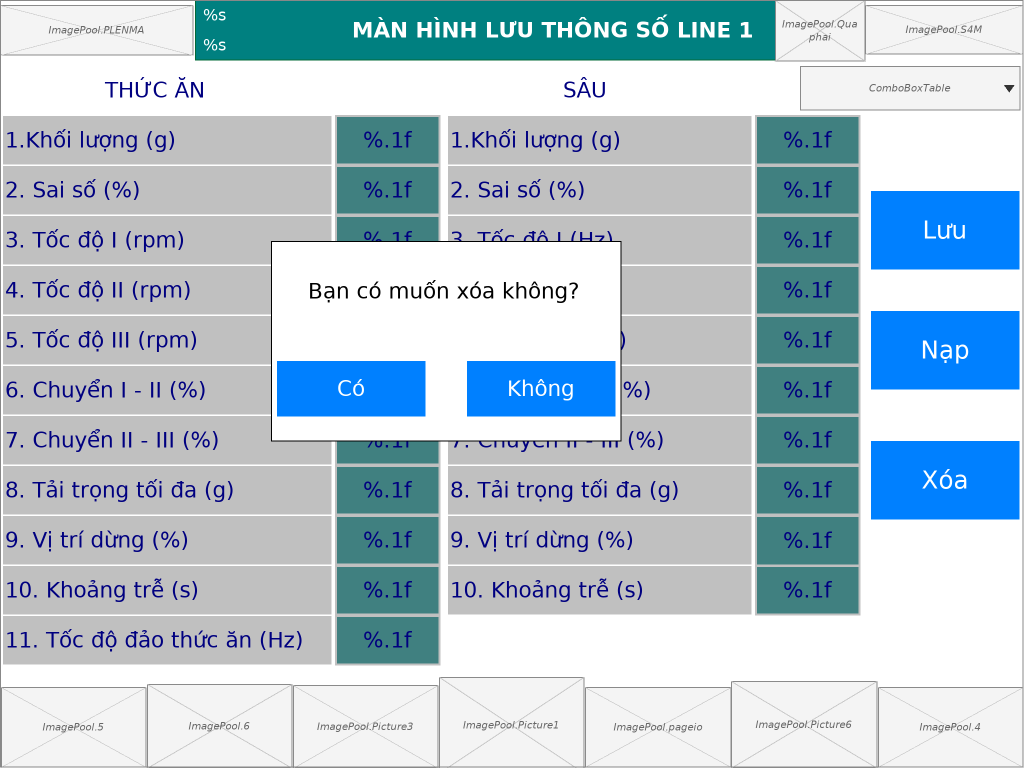
VISUALIZATION N_Recipe_Line1  // 1024x768
    Frame (0,687 1024x80)
        shows N_Footer_Line1()
    Frame (0,0 1024x60)
        shows N_Header()
    Textfield (353,5 400x50), "MÀN HÌNH LƯU THÔNG SỐ LINE 1"
    Textfield (80,75 150x30), "THỨC ĂN"
    Textfield (545,75 80x30), "SÂU"
    Rectangle (870,190 150x80), "Lưu"
        tap GVL_OF_VU.bRecSave[1]
        OnDialogClosed: execute { bSave1 := true; }
        OnMouseClick: write PRG_MainRecipe1.NameSave via VisuDialogs.Keypad
    Rectangle (870,440 150x80), "Xóa"
        tap GVL_OF_VU.bRecDelete[1]
        OnMouseDown: execute { GVL_OF_VU.bDeleteRecipe1 := TRUE; }
    Rectangle (870,310 150x80), "Nạp"
        tap GVL_OF_VU.bRecLoad[1]
        OnMouseDown: execute { bLoad1 := true; }
    ComboBoxTable (800,66 220x44), variable: PRG_MainRecipe1.RecipeNameIdx, data array: PRG_MainRecipe1.RecipeList
        p3854506369: PRG_MainRecipe1.RecipeList[INDEX]
    Rectangle (447,115 305x50), "1.Khối lượng (g)"
    Rectangle (447,165 305x50), "2. Sai số (%)"
    Rectangle (447,215 305x50), "3. Tốc độ I (Hz)"
    Rectangle (447,265 305x50), "4. Tốc độ II (Hz)"
    Rectangle (447,365 305x50), "6. Chuyển I - II (%)"
    Rectangle (447,465 305x50), "8. Tải trọng tối đa (g)"
    Rectangle (447,315 305x50), "5. Tốc độ III (Hz)"
    Rectangle (447,415 305x50), "7. Chuyển II - III (%)"
    Rectangle (447,565 305x50), "10. Khoảng trễ (s)"
    Rectangle (447,515 305x50), "9. Vị trí dừng (%)"
    Rectangle (2,115 330x50), "1.Khối lượng (g)"
    Rectangle (2,165 330x50), "2. Sai số (%)"
    Rectangle (2,215 330x50), "3. Tốc độ I (rpm)"
    Rectangle (2,265 330x50), "4. Tốc độ II (rpm)"
    Rectangle (2,365 330x50), "6. Chuyển I - II (%)"
    Rectangle (2,465 330x50), "8. Tải trọng tối đa (g)"
    Rectangle (2,315 330x50), "5. Tốc độ III (rpm)"
    Rectangle (2,415 330x50), "7. Chuyển II - III (%)"
    Rectangle (2,565 330x50), "10. Khoảng trễ (s)"
    Rectangle (2,515 330x50), "9. Vị trí dừng (%)"
    Rectangle (2,615 330x50), "11. Tốc độ đảo thức ăn (Hz)"
    Image (775,0 90x61), image: ImagePool.Qua phai
        OnMouseClick: change screen: N_Recipe_Line2
    Textfield (335,115 105x50), "%.1f", text variable: PR_Line01.fDerisedWeight_Food
    Textfield (335,165 105x50), "%.1f", text variable: PR_Line01.fDelta_Food
    Textfield (335,215 105x50), "%.1f", text variable: PR_Line01.fFast_Speed
    Textfield (335,265 105x50), "%.1f", text variable: PR_Line01.fSlow_Speed_1
    Textfield (335,315 105x50), "%.1f", text variable: PR_Line01.fSlow_Speed_2
    Textfield (335,365 105x50), "%.1f", text variable: PR_Line01.fChangeMode_Food_1
    Textfield (335,415 105x50), "%.1f", text variable: PR_Line01.fChangeMode_Food_2
    Textfield (335,465 105x50), "%.1f", text variable: PR_Line01.fMaxWeight_Food
    Textfield (335,515 105x50), "%.1f", text variable: PR_Line01.fPerStop_Food
    Textfield (335,565 105x50), "%.1f", text variable: PR_Line01.fTimer_Check_Food
    Textfield (335,615 105x50), "%.1f", text variable: PR_Line01.fSpeed_motor_mixer
    Textfield (755,115 105x50), "%.1f", text variable: PR_Line01.fDerisedWeight_Worm
    Textfield (755,165 105x50), "%.1f", text variable: PR_Line01.fDelta_Worm
    Textfield (755,215 105x50), "%.1f", text variable: PR_Line01.fFast_Speed_vibrating_funnel
    Textfield (755,265 105x50), "%.1f", text variable: PR_Line01.fSlow_Speed_vibrating_funnel_1
    Textfield (755,315 105x50), "%.1f", text variable: PR_Line01.fSlow_Speed_vibrating_funnel_2
    Textfield (755,365 105x50), "%.1f", text variable: PR_Line01.fChangeMode_Worm_1
    Textfield (755,415 105x50), "%.1f", text variable: PR_Line01.fChangeMode_Worm_2
    Textfield (755,465 105x50), "%.1f", text variable: PR_Line01.fMaxWeight_Worm
    Textfield (755,515 105x51), "%.1f", text variable: PR_Line01.fPerStop_Worm
    Textfield (755,565 105x50), "%.1f", text variable: PR_Line01.fTimer_Check_Worm
    GroupBox (271,241 350x200), invisible if: not GVL_OF_VU.bDeleteRecipe1, input disabled if: not GVL_OF_VU.bDeleteRecipe1
        Rectangle (0,0 350x200)
        Rectangle (5,119 150x57), "Có"
            OnMouseDown: execute { bDelete1 := true; }
            OnMouseUp: execute { GVL_OF_VU.bDeleteRecipe1 := FALSE; }
        Label (4,29 338x42), "Bạn có muốn xóa không?"
        Rectangle (195,119 150x57), "Không"
            OnMouseDown: execute { GVL_OF_VU.bDeleteRecipe1 := FALSE; }
END_VISUALIZATION

// ---- VISUs/Recipe/N_Recipe_Line2.TcVIS
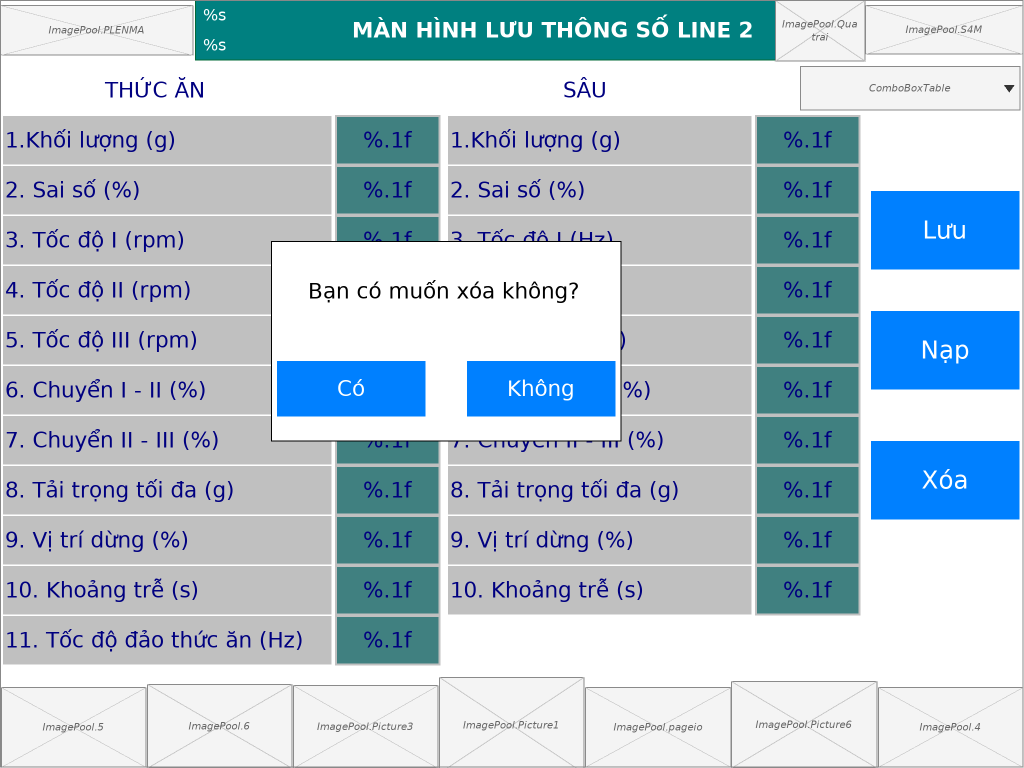
VISUALIZATION N_Recipe_Line2  // 1024x768
    Frame (0,687 1024x80)
        shows N_Footer_Line2()
    Frame (0,0 1024x60)
        shows N_Header()
    Textfield (353,5 400x50), "MÀN HÌNH LƯU THÔNG SỐ LINE 2"
    Textfield (80,75 150x30), "THỨC ĂN"
    Textfield (545,75 80x30), "SÂU"
    Rectangle (870,190 150x80), "Lưu"
        tap GVL_OF_VU.bRecSave[2]
        OnDialogClosed: execute { bSave2 := true; }
        OnMouseDown: write PRG_MainRecipe1_1.NameSave via VisuDialogs.Keypad
    Rectangle (870,440 150x80), "Xóa"
        tap GVL_OF_VU.bRecDelete[2]
        OnMouseClick: execute { GVL_OF_VU.bDeleteRecipe2 := true; }
    Rectangle (870,310 150x80), "Nạp"
        tap GVL_OF_VU.bRecLoad[2]
        OnMouseClick: execute { bLoad2 := true; }
    Group (447,115 305x500)
        Rectangle (0,0 305x50), "1.Khối lượng (g)"
        Rectangle (0,50 305x50), "2. Sai số (%)"
        Rectangle (0,100 305x50), "3. Tốc độ I (Hz)"
        Rectangle (0,150 305x50), "4. Tốc độ II (Hz)"
        Rectangle (0,250 305x50), "6. Chuyển I - II (%)"
        Rectangle (0,350 305x50), "8. Tải trọng tối đa (g)"
        Rectangle (0,200 305x50), "5. Tốc độ III (Hz)"
        Rectangle (0,300 305x50), "7. Chuyển II - III (%)"
        Rectangle (0,450 305x50), "10. Khoảng trễ (s)"
        Rectangle (0,400 305x50), "9. Vị trí dừng (%)"
    Textfield (755,115 105x50), "%.1f", text variable: PR_Line02.fDerisedWeight_Worm
    Textfield (755,165 105x50), "%.1f", text variable: PR_Line02.fDelta_Worm
    Textfield (755,215 105x50), "%.1f", text variable: PR_Line02.fFast_Speed_vibrating_funnel
    Textfield (755,265 105x50), "%.1f", text variable: PR_Line02.fSlow_Speed_vibrating_funnel_1
    Textfield (755,315 105x50), "%.1f", text variable: PR_Line02.fSlow_Speed_vibrating_funnel_2
    Textfield (755,365 105x50), "%.1f", text variable: PR_Line02.fChangeMode_Worm_1
    Textfield (755,415 105x50), "%.1f", text variable: PR_Line02.fChangeMode_Worm_2
        OnMouseDown: write GVL_OF_VU.fRecChangeII_IIIOfWorm[2] via VisuDialogs.Numpad
    Textfield (755,465 105x50), "%.1f", text variable: PR_Line02.fMaxWeight_Worm
    Textfield (755,515 105x50), "%.1f", text variable: PR_Line02.fPerStop_Worm
    Textfield (755,565 105x50), "%.1f", text variable: PR_Line02.fTimer_check_Worm
    Rectangle (2,115 330x50), "1.Khối lượng (g)"
    Rectangle (2,165 330x50), "2. Sai số (%)"
    Rectangle (2,215 330x50), "3. Tốc độ I (rpm)"
    Rectangle (2,265 330x50), "4. Tốc độ II (rpm)"
    Rectangle (2,365 330x50), "6. Chuyển I - II (%)"
    Rectangle (2,465 330x50), "8. Tải trọng tối đa (g)"
    Rectangle (2,315 330x50), "5. Tốc độ III (rpm)"
    Rectangle (2,415 330x50), "7. Chuyển II - III (%)"
    Rectangle (2,565 330x50), "10. Khoảng trễ (s)"
    Rectangle (2,515 330x50), "9. Vị trí dừng (%)"
    Rectangle (2,615 330x50), "11. Tốc độ đảo thức ăn (Hz)"
    Textfield (335,115 105x50), "%.1f", text variable: PR_Line02.fDerisedWeight_Food
    Textfield (335,165 105x50), "%.1f", text variable: PR_Line02.fDelta_Food
    Textfield (335,215 105x50), "%.1f", text variable: PR_Line02.fFast_Speed
    Textfield (335,265 105x50), "%.1f", text variable: PR_Line02.fSlow_Speed_1
    Textfield (335,315 105x50), "%.1f", text variable: PR_Line02.fSlow_Speed_2
    Textfield (335,365 105x50), "%.1f", text variable: PR_Line02.fChangeMode_Food_1
    Textfield (335,415 105x50), "%.1f", text variable: PR_Line02.fChangeMode_Food_2
    Textfield (335,465 105x50), "%.1f", text variable: PR_Line02.fMaxWeight_Food
    Textfield (335,515 105x50), "%.1f", text variable: PR_Line02.fPerStop_Food
    Textfield (335,565 105x50), "%.1f", text variable: PR_Line02.fTimer_Check_Food
    Textfield (335,615 105x50), "%.1f", text variable: PR_Line02.fSpeed_motor_mixer
    Image (775,0 90x61), image: ImagePool.Qua trai
        OnMouseClick: change screen: N_Recipe_Line1
    ComboBoxTable (800,66 220x44), variable: PRG_MainRecipe1_1.RecipeNameIdx, data array: PRG_MainRecipe1_1.RecipeList
        p3854506369: PRG_MainRecipe1_1.RecipeList[INDEX]
    GroupBox (271,241 350x200), invisible if: not GVL_OF_VU.bDeleteRecipe2, input disabled if: not GVL_OF_VU.bDeleteRecipe2
        Rectangle (0,0 350x200)
        Rectangle (5,119 150x57), "Có"
            OnMouseDown: execute { bDelete2 := true; }
            OnMouseUp: execute { GVL_OF_VU.bDeleteRecipe2 := FALSE; }
        Label (4,29 338x42), "Bạn có muốn xóa không?"
        Rectangle (195,119 150x57), "Không"
            OnMouseDown: execute { GVL_OF_VU.bDeleteRecipe2 := FALSE; }
END_VISUALIZATION

// ---- VISUs/Setting/N_Setting_Delay_FoodSupply1.TcVIS
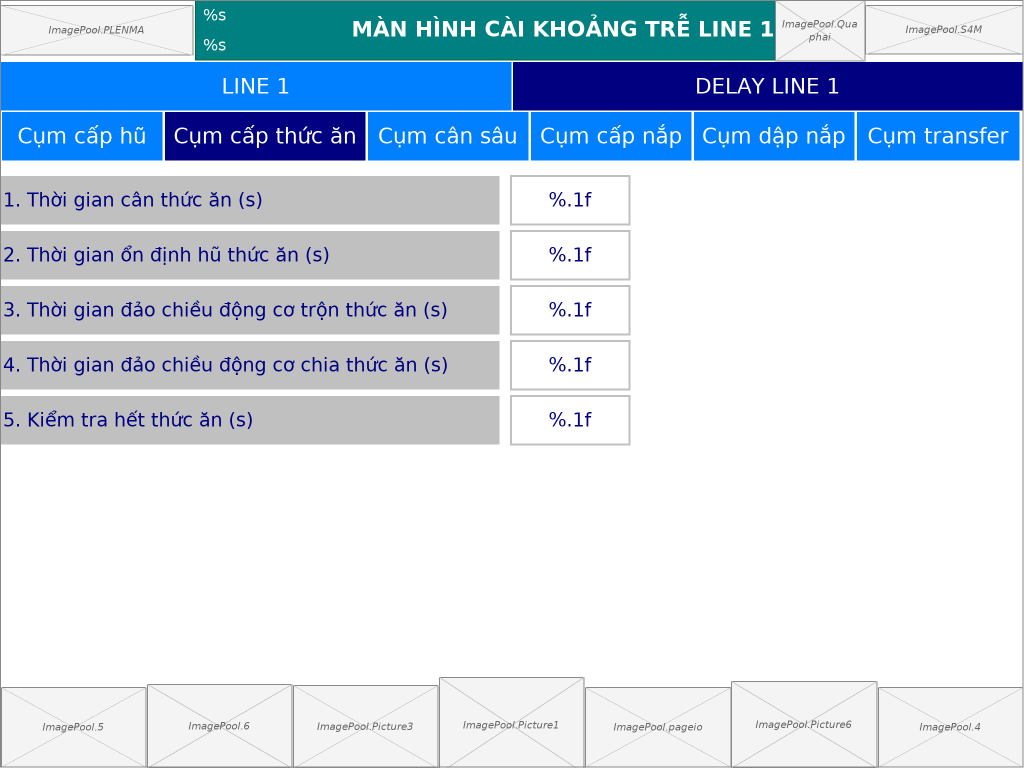
VISUALIZATION N_Setting_Delay_FoodSupply1  // 1024x768
    Frame (0,687 1024x80)
        shows N_Footer_Line1()
    Frame (0,0 1024x60)
        shows N_Header()
    Textfield (353,4 420x50), "MÀN HÌNH CÀI KHOẢNG TRỄ LINE 1"
    Rectangle (0,61 512x50), "LINE 1"
        OnMouseClick: change screen: N_Setting_Line1
    Rectangle (512,61 511x50), "DELAY LINE 1"
        OnMouseClick: change screen: N_Setting_Delay_JarSupply1
    Image (775,0 90x61), image: ImagePool.Qua phai
        OnMouseClick: change screen: N_Setting_Delay_FoodSupply2
    Rectangle (0,175 500x50), "1. Thời gian cân thức ăn (s)"
    Rectangle (510,175 120x50), "%.1f", text variable: PR_Line01.fTimer_Alarm_Food
        OnMouseClick: write PR_Line01.fTimer_Alarm_Food via VisuDialogs.Numpad
    Rectangle (0,230 500x50), "2. Thời gian ổn định hũ thức ăn (s)"
    Rectangle (510,230 120x50), "%.1f", text variable: PR_Line01.fTimer_Food
        OnMouseClick: write PR_Line01.fTimer_Food via VisuDialogs.Numpad
    Rectangle (0,285 500x50), "3. Thời gian đảo chiều động cơ trộn thức ăn (s)"
    Rectangle (0,340 500x50), "4. Thời gian đảo chiều động cơ chia thức ăn (s)"
    Rectangle (510,285 120x50), "%.1f", text variable: PR_Line01.fTimer_Reverse
        OnMouseClick: write PR_Line01.fTimer_Reverse via VisuDialogs.Numpad
    Rectangle (510,340 120x50), "%.1f", text variable: PR_Line01.fTimer_rever_food
        OnMouseClick: write PR_Line01.fTimer_rever_food via VisuDialogs.Numpad
    Rectangle (1,111 162x50), "Cụm cấp hũ"
        OnMouseClick: change screen: N_Setting_Delay_JarSupply1
    Rectangle (164,111 202x50), "Cụm cấp thức ăn"
        OnMouseClick: change screen: N_Setting_Delay_FoodSupply1
    Rectangle (367,111 162x50), "Cụm cân sâu"
        OnMouseClick: change screen: N_Setting_Delay_WormWeight1
    Rectangle (530,111 162x50), "Cụm cấp nắp"
        OnMouseClick: change screen: N_Setting_Delay_LidSupply1
    Rectangle (693,111 162x50), "Cụm dập nắp"
        OnMouseClick: change screen: N_Setting_Delay_LidPressing1
    Rectangle (856,111 164x50), "Cụm transfer"
        OnMouseClick: change screen: N_Setting_Delay_Tranfer1
    Rectangle (0,395 500x50), "5. Kiểm tra hết thức ăn (s)"
    Rectangle (510,395 120x50), "%.1f", text variable: PR_Line01.fTimer_Error_Food
        OnMouseClick: write PR_Line01.fTimer_Error_Food via VisuDialogs.Numpad
END_VISUALIZATION

// ---- VISUs/Setting/N_Setting_Delay_FoodSupply2.TcVIS
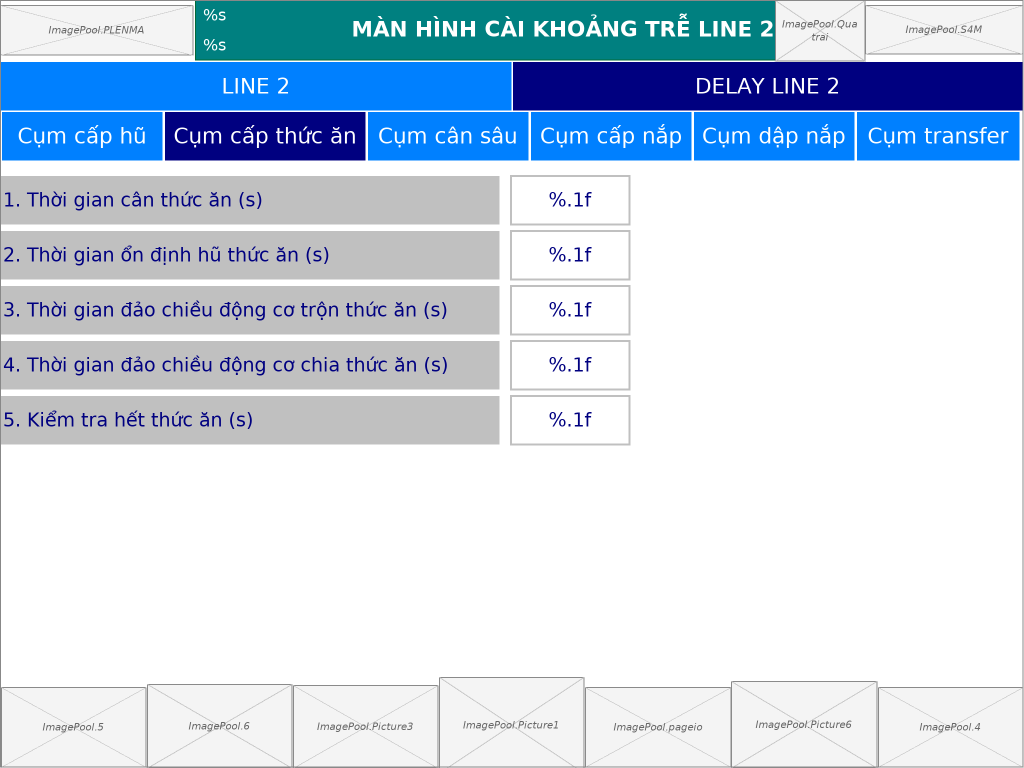
VISUALIZATION N_Setting_Delay_FoodSupply2  // 1024x768
    Frame (0,687 1024x80)
        shows N_Footer_Line2()
    Frame (0,0 1024x60)
        shows N_Header()
    Textfield (353,4 420x50), "MÀN HÌNH CÀI KHOẢNG TRỄ LINE 2"
    Rectangle (0,175 500x50), "1. Thời gian cân thức ăn (s)"
    Rectangle (0,230 500x50), "2. Thời gian ổn định hũ thức ăn (s)"
    Rectangle (0,285 500x50), "3. Thời gian đảo chiều động cơ trộn thức ăn (s)"
    Rectangle (0,340 500x50), "4. Thời gian đảo chiều động cơ chia thức ăn (s)"
    Rectangle (0,61 512x50), "LINE 2"
        OnMouseClick: change screen: N_Setting_Line2
    Rectangle (1,111 162x50), "Cụm cấp hũ"
        OnMouseClick: change screen: N_Setting_Delay_JarSupply2
    Rectangle (164,111 202x50), "Cụm cấp thức ăn"
        OnMouseClick: change screen: N_Setting_Delay_FoodSupply2
    Rectangle (367,111 162x50), "Cụm cân sâu"
        OnMouseClick: change screen: N_Setting_Delay_WorwWeight2
    Rectangle (530,111 162x50), "Cụm cấp nắp"
        OnMouseClick: change screen: N_Setting_Delay_LidSupply2
    Rectangle (693,111 162x50), "Cụm dập nắp"
        OnMouseClick: change screen: N_Setting_Delay_LidPressing2
    Rectangle (856,111 164x50), "Cụm transfer"
        OnMouseClick: change screen: N_Setting_Delay_Tranfer2
    Rectangle (512,61 511x50), "DELAY LINE 2"
        OnMouseClick: change screen: N_Setting_Delay_JarSupply2
    Image (775,0 90x61), image: ImagePool.Qua trai
        OnMouseClick: change screen: N_Setting_Delay_FoodSupply1
    Rectangle (510,175 120x50), "%.1f", text variable: PR_Line02.fTimer_Alarm_Food
        OnMouseClick: write PR_Line02.fTimer_Alarm_Food via VisuDialogs.Numpad
    Rectangle (510,230 120x50), "%.1f", text variable: PR_Line02.fTimer_Food
        OnMouseClick: write PR_Line02.fTimer_Food via VisuDialogs.Numpad
    Rectangle (510,285 120x50), "%.1f", text variable: PR_Line02.fTimer_Reverse
        OnMouseClick: write PR_Line02.fTimer_Reverse via VisuDialogs.Numpad
    Rectangle (510,340 120x50), "%.1f", text variable: PR_Line02.fTimer_rever_food
        OnMouseClick: write PR_Line02.fTimer_rever_food via VisuDialogs.Numpad
    Rectangle (0,395 500x50), "5. Kiểm tra hết thức ăn (s)"
    Rectangle (510,395 120x50), "%.1f", text variable: PR_Line02.fTimer_Error_Food
        OnMouseClick: write PR_Line02.fTimer_Error_Food via VisuDialogs.Numpad
END_VISUALIZATION

// ---- VISUs/Setting/N_Setting_Delay_JarSupply1.TcVIS
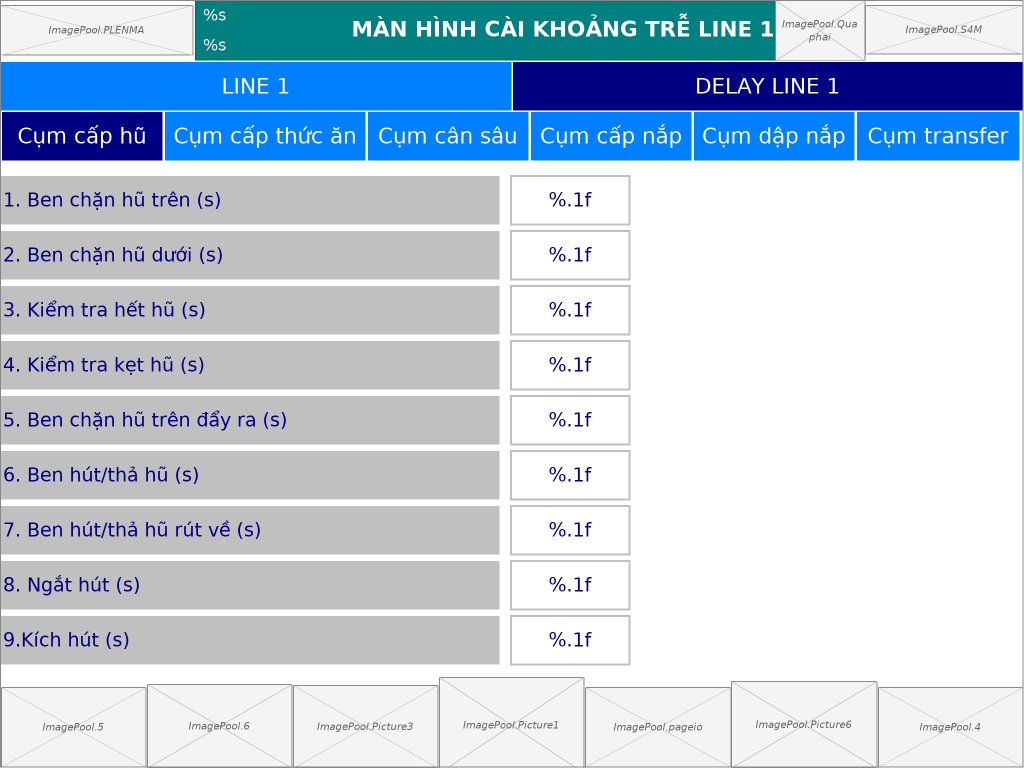
VISUALIZATION N_Setting_Delay_JarSupply1  // 1024x768
    Frame (0,687 1024x80)
        shows N_Footer_Line1()
    Frame (0,0 1024x60)
        shows N_Header()
    Textfield (353,4 420x50), "MÀN HÌNH CÀI KHOẢNG TRỄ LINE 1"
    Rectangle (0,61 512x50), "LINE 1"
        OnMouseClick: change screen: N_Setting_Line1
    Image (775,0 90x61), image: ImagePool.Qua phai
        OnMouseClick: change screen: N_Setting_Delay_JarSupply2
    Rectangle (1,111 162x50), "Cụm cấp hũ"
        OnMouseClick: change screen: N_Setting_Delay_JarSupply1
    Rectangle (164,111 202x50), "Cụm cấp thức ăn"
        OnMouseClick: change screen: N_Setting_Delay_FoodSupply1
    Rectangle (367,111 162x50), "Cụm cân sâu"
        OnMouseClick: change screen: N_Setting_Delay_WormWeight1
    Rectangle (530,111 162x50), "Cụm cấp nắp"
        OnMouseClick: change screen: N_Setting_Delay_LidSupply1
    Rectangle (693,111 162x50), "Cụm dập nắp"
        OnMouseClick: change screen: N_Setting_Delay_LidPressing1
    Rectangle (856,111 164x50), "Cụm transfer"
        OnMouseClick: change screen: N_Setting_Delay_Tranfer1
    Rectangle (512,61 511x50), "DELAY LINE 1"
        OnMouseClick: change screen: N_Setting_Delay_JarSupply1
    Rectangle (0,175 500x50), "1. Ben chặn hũ trên (s)"
    Rectangle (510,175 120x50), "%.1f", text variable: PR_Line01.timerCheckCylinder_Up
        OnMouseClick: write PR_Line01.timerCheckCylinder_Up via VisuDialogs.Numpad
    Rectangle (0,230 500x50), "2. Ben chặn hũ dưới (s)"
    Rectangle (510,230 120x50), "%.1f", text variable: PR_Line01.timerCheckCylinder_Dw
        OnMouseClick: write PR_Line01.timerCheckCylinder_Dw via VisuDialogs.Numpad
    Rectangle (0,340 500x50), "4. Kiểm tra kẹt hũ (s)"
    Rectangle (0,285 500x50), "3. Kiểm tra hết hũ (s)"
    Rectangle (510,285 120x50), "%.1f", text variable: PR_Line01.timerCheckEmpty
        OnMouseClick: write PR_Line01.timerCheckEmpty via VisuDialogs.Numpad
    Rectangle (510,340 120x50), "%.1f", text variable: PR_Line01.timerCheckStuck
        OnMouseClick: write PR_Line01.timerCheckStuck via VisuDialogs.Numpad
    Rectangle (0,395 500x50), "5. Ben chặn hũ trên đẩy ra (s)"
    Rectangle (510,395 120x50), "%.1f", text variable: PR_Line01.timerCylinder_Up_extend
        OnMouseClick: write PR_Line01.timerCylinder_Up_extend via VisuDialogs.Numpad
    Rectangle (0,450 500x50), "6. Ben hút/thả hũ (s)"
    Rectangle (510,450 120x50), "%.1f", text variable: PR_Line01.timerCylinder_Suction_Cup
        OnMouseClick: write PR_Line01.timerCylinder_Suction_Cup via VisuDialogs.Numpad
    Rectangle (0,505 500x50), "7. Ben hút/thả hũ rút về (s)"
    Rectangle (510,505 120x50), "%.1f", text variable: PR_Line01.timerCylinder_Suction_Cup_extend
        OnMouseClick: write PR_Line01.timerCylinder_Suction_Cup_extend via VisuDialogs.Numpad
    Rectangle (0,560 500x50), "8. Ngắt hút (s)"
    Rectangle (510,560 120x50), "%.1f", text variable: PR_Line01.timerCylinder_Suction_Val
        OnMouseClick: write PR_Line01.timerCylinder_Suction_Val via VisuDialogs.Numpad
    Rectangle (0,615 500x50), "9.Kích hút (s)"
    Rectangle (510,615 120x50), "%.1f", text variable: PR_Line01.timerCylinder_Suction_pick
        OnMouseClick: write PR_Line01.timerCylinder_Suction_pick via VisuDialogs.Numpad
END_VISUALIZATION

// ---- VISUs/Setting/N_Setting_Delay_JarSupply2.TcVIS
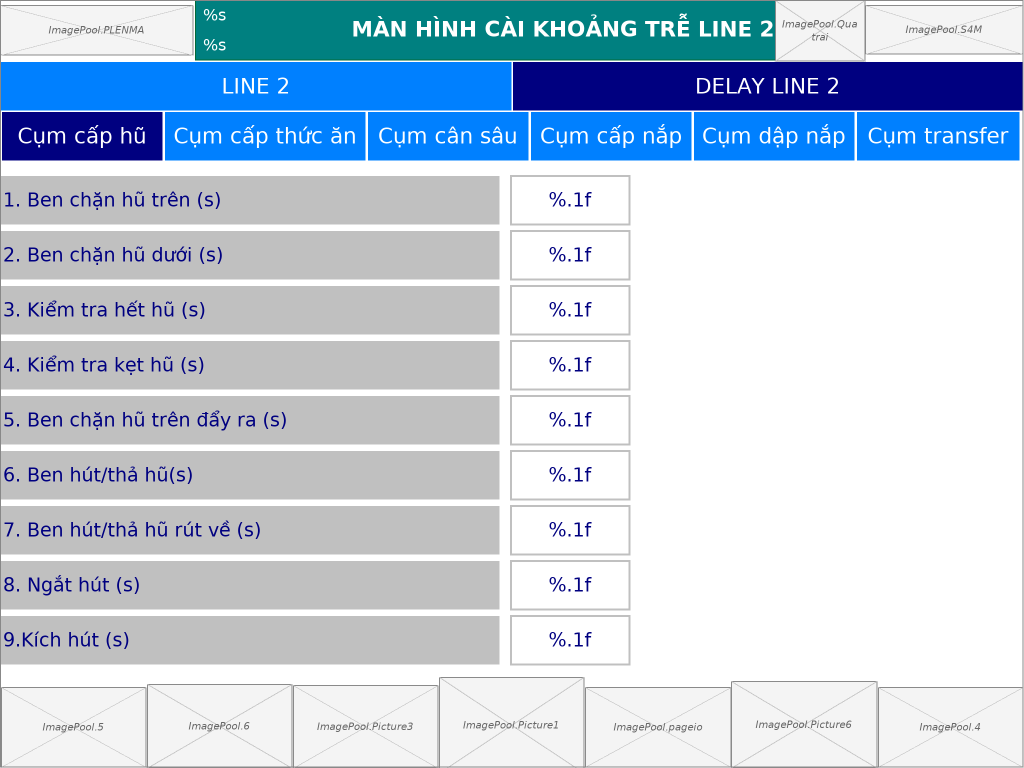
VISUALIZATION N_Setting_Delay_JarSupply2  // 1024x768
    Frame (0,687 1024x80)
        shows N_Footer_Line2()
    Frame (0,0 1024x60)
        shows N_Header()
    Textfield (353,4 420x50), "MÀN HÌNH CÀI KHOẢNG TRỄ LINE 2"
    Rectangle (0,175 500x50), "1. Ben chặn hũ trên (s)"
    Rectangle (0,230 500x50), "2. Ben chặn hũ dưới (s)"
    Rectangle (0,340 500x50), "4. Kiểm tra kẹt hũ (s)"
    Rectangle (0,285 500x50), "3. Kiểm tra hết hũ (s)"
    Rectangle (0,395 500x50), "5. Ben chặn hũ trên đẩy ra (s)"
    Rectangle (0,61 512x50), "LINE 2"
        OnMouseClick: change screen: N_Setting_Line2
    Rectangle (1,111 162x50), "Cụm cấp hũ"
        OnMouseClick: change screen: N_Setting_Delay_JarSupply2
    Rectangle (164,111 202x50), "Cụm cấp thức ăn"
        OnMouseClick: change screen: N_Setting_Delay_FoodSupply2
    Rectangle (367,111 162x50), "Cụm cân sâu"
        OnMouseClick: change screen: N_Setting_Delay_WorwWeight2
    Rectangle (530,111 162x50), "Cụm cấp nắp"
        OnMouseClick: change screen: N_Setting_Delay_LidSupply2
    Rectangle (693,111 162x50), "Cụm dập nắp"
        OnMouseClick: change screen: N_Setting_Delay_LidPressing2
    Rectangle (856,111 164x50), "Cụm transfer"
        OnMouseClick: change screen: N_Setting_Delay_Tranfer2
    Rectangle (512,61 511x50), "DELAY LINE 2"
        OnMouseClick: change screen: N_Setting_Delay_JarSupply2
    Image (775,0 90x61), image: ImagePool.Qua trai
        OnMouseClick: change screen: N_Setting_Delay_JarSupply1
    Rectangle (510,175 120x50), "%.1f", text variable: PR_Line02.timerCheckCylinder_Up
        OnMouseClick: write PR_Line02.timerCheckCylinder_Up via VisuDialogs.Numpad
    Rectangle (510,230 120x50), "%.1f", text variable: PR_Line02.timerCheckCylinder_Dw
        OnMouseClick: write PR_Line02.timerCheckCylinder_Dw via VisuDialogs.Numpad
    Rectangle (510,285 120x50), "%.1f", text variable: PR_Line02.timerCheckEmpty
        OnMouseClick: write PR_Line02.timerCheckEmpty via VisuDialogs.Numpad
    Rectangle (510,340 120x50), "%.1f", text variable: PR_Line02.timerCheckStuck
        OnMouseClick: write PR_Line02.timerCheckStuck via VisuDialogs.Numpad
    Rectangle (510,395 120x50), "%.1f", text variable: PR_Line02.timerCylinder_Up_extend
        OnMouseClick: write PR_Line02.timerCylinder_Up_extend via VisuDialogs.Numpad
    Rectangle (0,450 500x50), "6. Ben hút/thả hũ(s)"
    Rectangle (510,450 120x50), "%.1f", text variable: PR_Line02.timerCylinder_Suction_Cup
        OnMouseClick: write PR_Line02.timerCylinder_Suction_Cup via VisuDialogs.Numpad
    Rectangle (0,505 500x50), "7. Ben hút/thả hũ rút về (s)"
    Rectangle (510,505 120x50), "%.1f", text variable: PR_Line02.timerCylinder_Suction_Cup_extend
        OnMouseClick: write PR_Line02.timerCylinder_Suction_Cup_extend via VisuDialogs.Numpad
    Rectangle (0,560 500x50), "8. Ngắt hút (s)"
    Rectangle (510,560 120x50), "%.1f", text variable: PR_Line02.timerCylinder_Suction_Val
        OnMouseClick: write PR_Line02.timerCylinder_Suction_Val via VisuDialogs.Numpad
    Rectangle (0,615 500x50), "9.Kích hút (s)"
    Rectangle (510,615 120x50), "%.1f", text variable: PR_Line02.timerCylinder_Suction_pick
        OnMouseClick: write PR_Line02.timerCylinder_Suction_pick via VisuDialogs.Numpad
END_VISUALIZATION

// ---- VISUs/Setting/N_Setting_Delay_LidPressing1.TcVIS
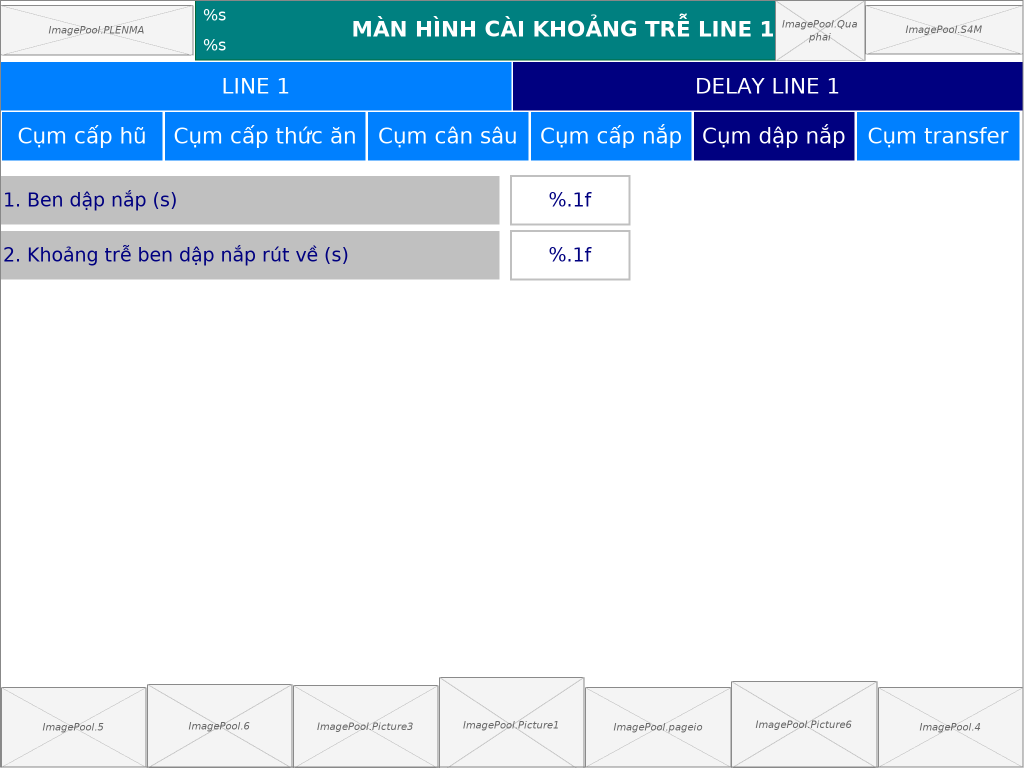
VISUALIZATION N_Setting_Delay_LidPressing1  // 1024x768
    Frame (0,687 1024x80)
        shows N_Footer_Line1()
    Frame (0,0 1024x60)
        shows N_Header()
    Textfield (353,4 420x50), "MÀN HÌNH CÀI KHOẢNG TRỄ LINE 1"
    Rectangle (0,61 512x50), "LINE 1"
        OnMouseClick: change screen: N_Setting_Line1
    Image (775,0 90x61), image: ImagePool.Qua phai
        OnMouseClick: change screen: N_Setting_Delay_LidPressing2
    Rectangle (0,175 500x50), "1. Ben dập nắp (s)"
    Rectangle (0,230 500x50), "2. Khoảng trễ ben dập nắp rút về (s)"
    Rectangle (510,175 120x50), "%.1f", text variable: PR_Line01.timer_Check_Cylinder_extend
        OnMouseClick: write PR_Line01.timer_Check_Cylinder_extend via VisuDialogs.Numpad
    Rectangle (510,230 120x50), "%.1f", text variable: PR_Line01.timer_Check_Cylinder_retract
        OnMouseClick: write PR_Line01.timer_Check_Cylinder_retract via VisuDialogs.Numpad
    Rectangle (1,111 162x50), "Cụm cấp hũ"
        OnMouseClick: change screen: N_Setting_Delay_JarSupply1
    Rectangle (164,111 202x50), "Cụm cấp thức ăn"
        OnMouseClick: change screen: N_Setting_Delay_FoodSupply1
    Rectangle (367,111 162x50), "Cụm cân sâu"
        OnMouseClick: change screen: N_Setting_Delay_WormWeight1
    Rectangle (530,111 162x50), "Cụm cấp nắp"
        OnMouseClick: change screen: N_Setting_Delay_LidSupply1
    Rectangle (693,111 162x50), "Cụm dập nắp"
        OnMouseClick: change screen: N_Setting_Delay_LidPressing1
    Rectangle (856,111 164x50), "Cụm transfer"
        OnMouseClick: change screen: N_Setting_Delay_Tranfer1
    Rectangle (512,61 511x50), "DELAY LINE 1"
        OnMouseClick: change screen: N_Setting_Delay_JarSupply1
END_VISUALIZATION

// ---- VISUs/Setting/N_Setting_Delay_LidPressing2.TcVIS
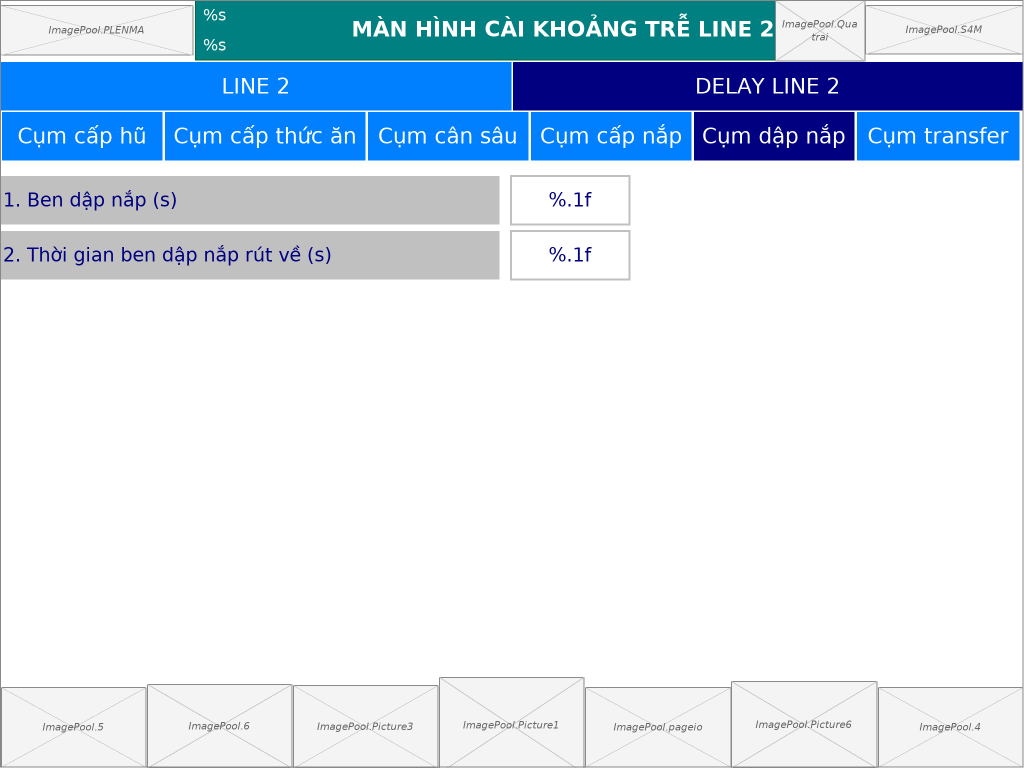
VISUALIZATION N_Setting_Delay_LidPressing2  // 1024x768
    Frame (0,687 1024x80)
        shows N_Footer_Line2()
    Frame (0,0 1024x60)
        shows N_Header()
    Textfield (353,4 420x50), "MÀN HÌNH CÀI KHOẢNG TRỄ LINE 2"
    Rectangle (0,175 500x50), "1. Ben dập nắp (s)"
    Rectangle (0,230 500x50), "2. Thời gian ben dập nắp rút về (s)"
    Rectangle (0,61 512x50), "LINE 2"
        OnMouseClick: change screen: N_Setting_Line2
    Rectangle (1,111 162x50), "Cụm cấp hũ"
        OnMouseClick: change screen: N_Setting_Delay_JarSupply2
    Rectangle (164,111 202x50), "Cụm cấp thức ăn"
        OnMouseClick: change screen: N_Setting_Delay_FoodSupply2
    Rectangle (367,111 162x50), "Cụm cân sâu"
        OnMouseClick: change screen: N_Setting_Delay_WorwWeight2
    Rectangle (530,111 162x50), "Cụm cấp nắp"
        OnMouseClick: change screen: N_Setting_Delay_LidSupply2
    Rectangle (693,111 162x50), "Cụm dập nắp"
        OnMouseClick: change screen: N_Setting_Delay_LidPressing2
    Rectangle (856,111 164x50), "Cụm transfer"
        OnMouseClick: change screen: N_Setting_Delay_Tranfer2
    Rectangle (512,61 511x50), "DELAY LINE 2"
        OnMouseClick: change screen: N_Setting_Delay_JarSupply2
    Image (775,0 90x61), image: ImagePool.Qua trai
        OnMouseClick: change screen: N_Setting_Delay_LidPressing1
    Rectangle (510,175 120x50), "%.1f", text variable: PR_Line02.timer_Check_Cylinder_extend
        OnMouseClick: write PR_Line02.timer_Check_Cylinder_extend via VisuDialogs.Numpad
    Rectangle (510,230 120x50), "%.1f", text variable: PR_Line02.timer_Check_Cylinder_retract
        OnMouseClick: write PR_Line02.timer_Check_Cylinder_retract via VisuDialogs.Numpad
END_VISUALIZATION

// ---- VISUs/Setting/N_Setting_Delay_LidSupply1.TcVIS
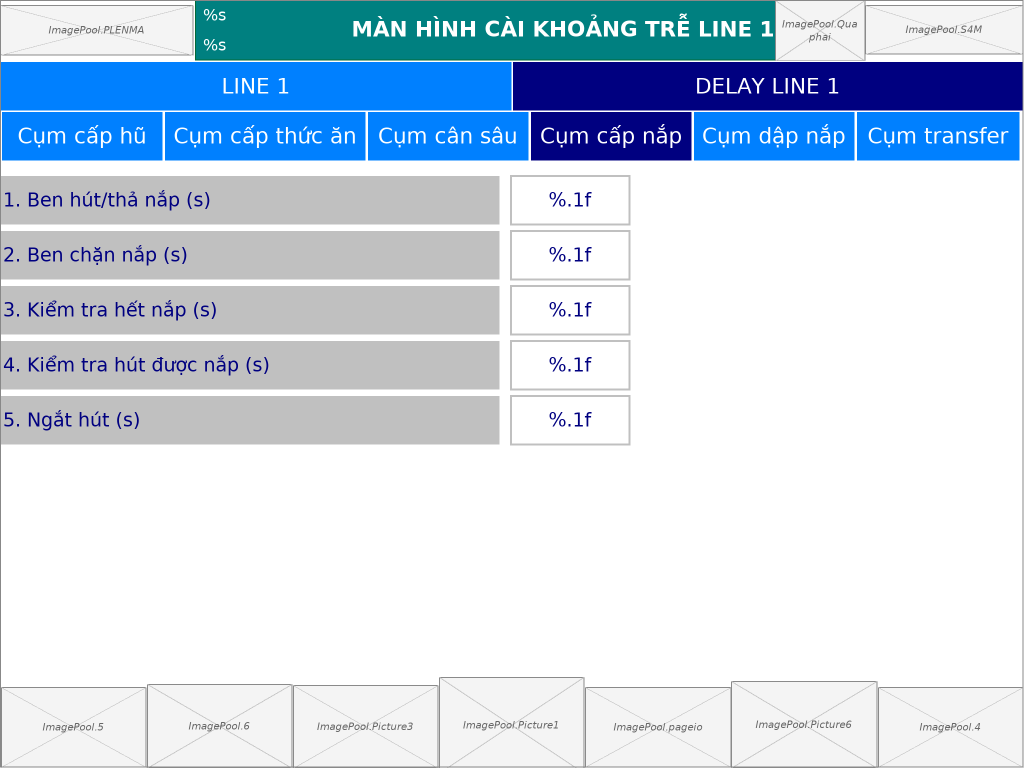
VISUALIZATION N_Setting_Delay_LidSupply1  // 1024x768
    Frame (0,687 1024x80)
        shows N_Footer_Line1()
    Frame (0,0 1024x60)
        shows N_Header()
    Textfield (353,4 420x50), "MÀN HÌNH CÀI KHOẢNG TRỄ LINE 1"
    Rectangle (0,61 512x50), "LINE 1"
        OnMouseClick: change screen: N_Setting_Line1
    Rectangle (1,111 162x50), "Cụm cấp hũ"
        OnMouseClick: change screen: N_Setting_Delay_JarSupply1
    Rectangle (164,111 202x50), "Cụm cấp thức ăn"
        OnMouseClick: change screen: N_Setting_Delay_FoodSupply1
    Rectangle (367,111 162x50), "Cụm cân sâu"
        OnMouseClick: change screen: N_Setting_Delay_WormWeight1
    Rectangle (530,111 162x50), "Cụm cấp nắp"
        OnMouseClick: change screen: N_Setting_Delay_LidSupply1
    Rectangle (693,111 162x50), "Cụm dập nắp"
        OnMouseClick: change screen: N_Setting_Delay_LidPressing1
    Rectangle (856,111 164x50), "Cụm transfer"
        OnMouseClick: change screen: N_Setting_Delay_Tranfer1
    Image (775,0 90x61), image: ImagePool.Qua phai
        OnMouseClick: change screen: N_Setting_Delay_LidSupply2
    Rectangle (0,175 500x50), "1. Ben hút/thả nắp (s)"
    Rectangle (0,230 500x50), "2. Ben chặn nắp (s)"
    Rectangle (510,175 120x50), "%.1f", text variable: PR_Line01.timerCylinder_Suction
        OnMouseClick: write PR_Line01.timerCylinder_Suction via VisuDialogs.Numpad
    Rectangle (0,285 500x50), "3. Kiểm tra hết nắp (s)"
    Rectangle (510,285 120x50), "%.1f", text variable: PR_Line01.timerCheckLidEmpty
        OnMouseClick: write PR_Line01.timerCheckLidEmpty via VisuDialogs.Numpad
    Rectangle (510,340 120x50), "%.1f", text variable: PR_Line01.timerCheckLidSuck
        OnMouseClick: write PR_Line01.timerCheckLidSuck via VisuDialogs.Numpad
    Rectangle (510,230 120x50), "%.1f", text variable: PR_Line01.timerCylinder_Stopper
        OnMouseClick: write PR_Line01.timerCylinder_Stopper via VisuDialogs.Numpad
    Rectangle (512,61 511x50), "DELAY LINE 1"
        OnMouseClick: change screen: N_Setting_Delay_JarSupply1
    Rectangle (0,340 500x50), "4. Kiểm tra hút được nắp (s)"
    Rectangle (510,395 120x50), "%.1f", text variable: PR_Line01.timerCheckLidRelease
        OnMouseClick: write PR_Line01.timerCheckLidRelease via VisuDialogs.Numpad
    Rectangle (0,395 500x50), "5. Ngắt hút (s)"
END_VISUALIZATION

// ---- VISUs/Setting/N_Setting_Delay_LidSupply2.TcVIS
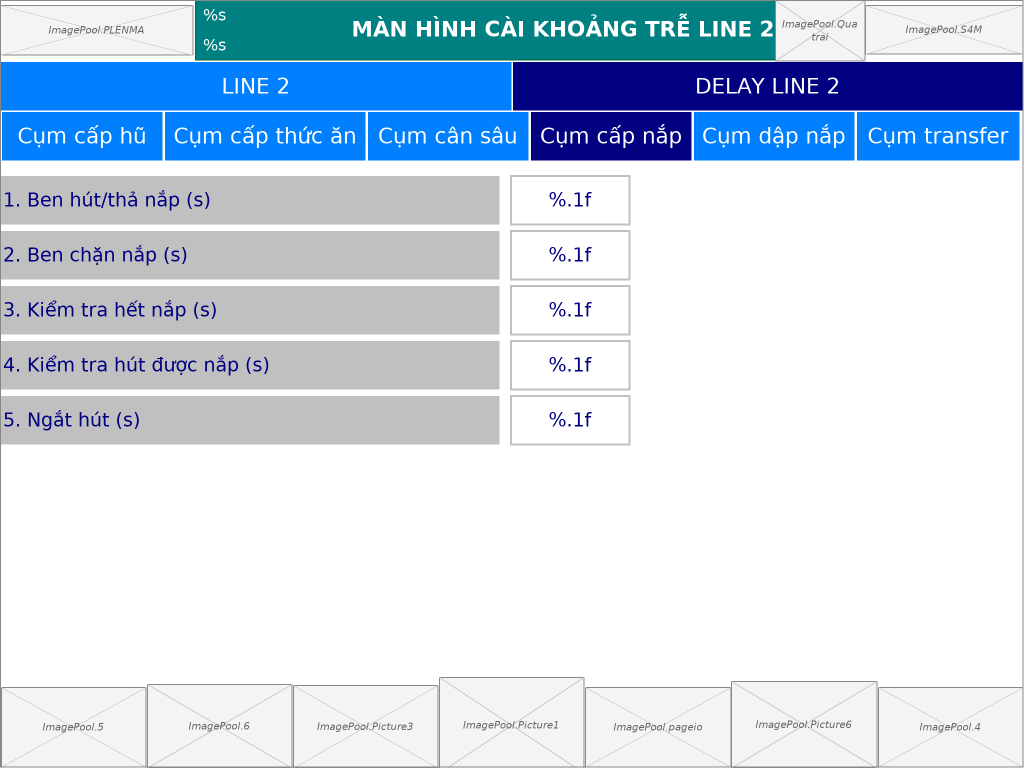
VISUALIZATION N_Setting_Delay_LidSupply2  // 1024x768
    Frame (0,687 1024x80)
        shows N_Footer_Line2()
    Frame (0,0 1024x60)
        shows N_Header()
    Textfield (353,4 420x50), "MÀN HÌNH CÀI KHOẢNG TRỄ LINE 2"
    Rectangle (0,175 500x50), "1. Ben hút/thả nắp (s)"
    Rectangle (0,340 500x50), "4. Kiểm tra hút được nắp (s)"
    Rectangle (0,230 500x50), "2. Ben chặn nắp (s)"
    Rectangle (0,285 500x50), "3. Kiểm tra hết nắp (s)"
    Rectangle (0,61 512x50), "LINE 2"
        OnMouseClick: change screen: N_Setting_Line2
    Rectangle (1,111 162x50), "Cụm cấp hũ"
        OnMouseClick: change screen: N_Setting_Delay_JarSupply2
    Rectangle (164,111 202x50), "Cụm cấp thức ăn"
        OnMouseClick: change screen: N_Setting_Delay_FoodSupply2
    Rectangle (367,111 162x50), "Cụm cân sâu"
        OnMouseClick: change screen: N_Setting_Delay_WorwWeight2
    Rectangle (530,111 162x50), "Cụm cấp nắp"
        OnMouseClick: change screen: N_Setting_Delay_LidSupply2
    Rectangle (693,111 162x50), "Cụm dập nắp"
        OnMouseClick: change screen: N_Setting_Delay_LidPressing2
    Rectangle (856,111 164x50), "Cụm transfer"
        OnMouseClick: change screen: N_Setting_Delay_Tranfer2
    Rectangle (512,61 511x50), "DELAY LINE 2"
        OnMouseClick: change screen: N_Setting_Delay_JarSupply2
    Image (775,0 90x61), image: ImagePool.Qua trai
        OnMouseClick: change screen: N_Setting_Delay_LidSupply1
    Rectangle (510,175 120x50), "%.1f", text variable: PR_Line02.timerCylinder_Suction
        OnMouseClick: write PR_Line02.timerCylinder_Suction via VisuDialogs.Numpad
    Rectangle (510,285 120x50), "%.1f", text variable: PR_Line02.timerCheckLidEmpty
        OnMouseClick: write PR_Line02.timerCheckLidEmpty via VisuDialogs.Numpad
    Rectangle (510,340 120x50), "%.1f", text variable: PR_Line02.timerCheckLidSuck
        OnMouseClick: write PR_Line02.timerCheckLidSuck via VisuDialogs.Numpad
    Rectangle (510,230 120x50), "%.1f", text variable: PR_Line02.timerCylinder_Stopper
        OnMouseClick: write PR_Line02.timerCylinder_Stopper via VisuDialogs.Numpad
    Rectangle (510,395 120x50), "%.1f", text variable: PR_Line02.timerCheckLidRelease
        OnMouseClick: write PR_Line02.timerCheckLidRelease via VisuDialogs.Numpad
    Rectangle (0,395 500x50), "5. Ngắt hút (s)"
END_VISUALIZATION

// ---- VISUs/Setting/N_Setting_Delay_Tranfer1.TcVIS
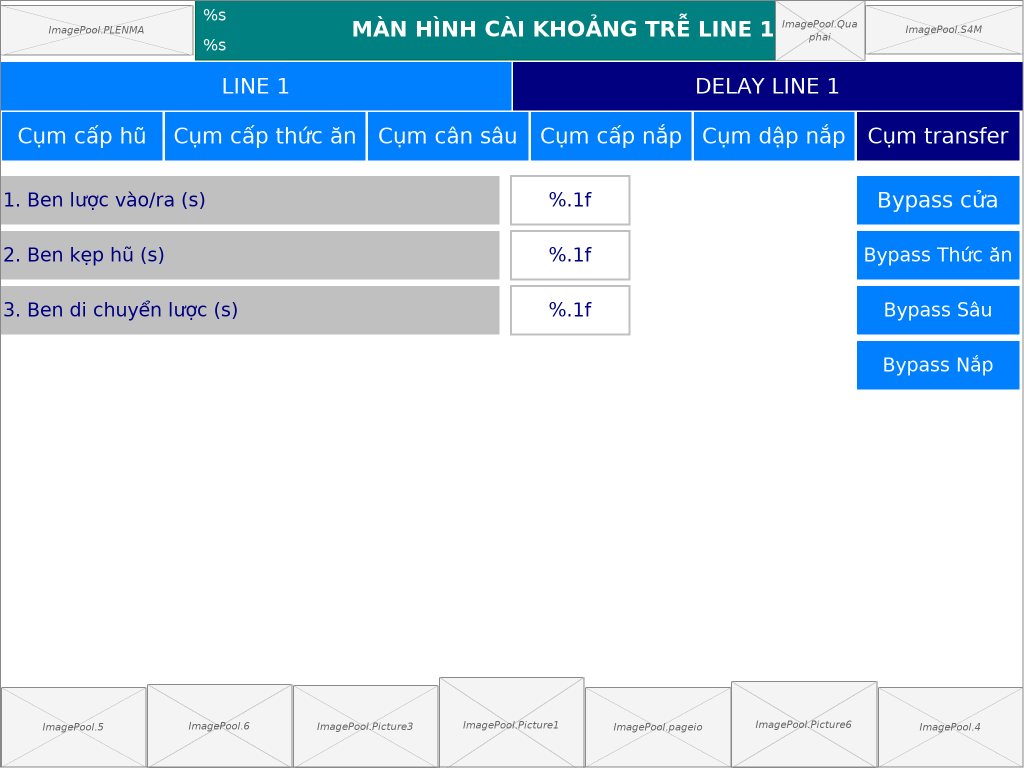
VISUALIZATION N_Setting_Delay_Tranfer1  // 1024x768
    Frame (0,687 1024x80)
        shows N_Footer_Line1()
    Frame (0,0 1024x60)
        shows N_Header()
    Textfield (353,4 420x50), "MÀN HÌNH CÀI KHOẢNG TRỄ LINE 1"
    Rectangle (0,61 512x50), "LINE 1"
        OnMouseClick: change screen: N_Setting_Line1
    Image (775,0 90x61), image: ImagePool.Qua phai
        OnMouseClick: change screen: N_Setting_Delay_Tranfer2
    Rectangle (0,230 500x50), "2. Ben kẹp hũ (s)"
    Rectangle (0,285 500x50), "3. Ben di chuyển lược (s)"
    Rectangle (510,175 120x50), "%.1f", text variable: PR_Line01.fTimer_Comb
        OnMouseClick: write PR_Line01.fTimer_Comb via VisuDialogs.Numpad
    Rectangle (510,230 120x50), "%.1f", text variable: PR_Line01.fTimer_Clip
        OnMouseClick: write PR_Line01.fTimer_Clip via VisuDialogs.Numpad
    Rectangle (510,285 120x50), "%.1f", text variable: PR_Line01.fTimer_Move_Comb
        OnMouseClick: write PR_Line01.fTimer_Move_Comb via VisuDialogs.Numpad
    Rectangle (1,111 162x50), "Cụm cấp hũ"
        OnMouseClick: change screen: N_Setting_Delay_JarSupply1
    Rectangle (164,111 202x50), "Cụm cấp thức ăn"
        OnMouseClick: change screen: N_Setting_Delay_FoodSupply1
    Rectangle (367,111 162x50), "Cụm cân sâu"
        OnMouseClick: change screen: N_Setting_Delay_WormWeight1
    Rectangle (530,111 162x50), "Cụm cấp nắp"
        OnMouseClick: change screen: N_Setting_Delay_LidSupply1
    Rectangle (693,111 162x50), "Cụm dập nắp"
        OnMouseClick: change screen: N_Setting_Delay_LidPressing1
    Rectangle (856,111 164x50), "Cụm transfer"
        OnMouseClick: change screen: N_Setting_Delay_Tranfer1
    Rectangle (512,61 511x50), "DELAY LINE 1"
        OnMouseClick: change screen: N_Setting_Delay_JarSupply1
    Rectangle (0,175 500x50), "1. Ben lược vào/ra (s)"
    Rectangle (856,175 164x50), "Bypass cửa"
        toggle bypass
    Rectangle (856,230 164x50), "Bypass Thức ăn"
        toggle PR_Line01.bypassfood
    Rectangle (856,285 164x50), "Bypass Sâu"
        toggle PR_Line01.bypassWorm
    Rectangle (856,340 164x50), "Bypass Nắp"
        toggle PR_Line01.bypassLid
END_VISUALIZATION

// ---- VISUs/Setting/N_Setting_Delay_Tranfer2.TcVIS
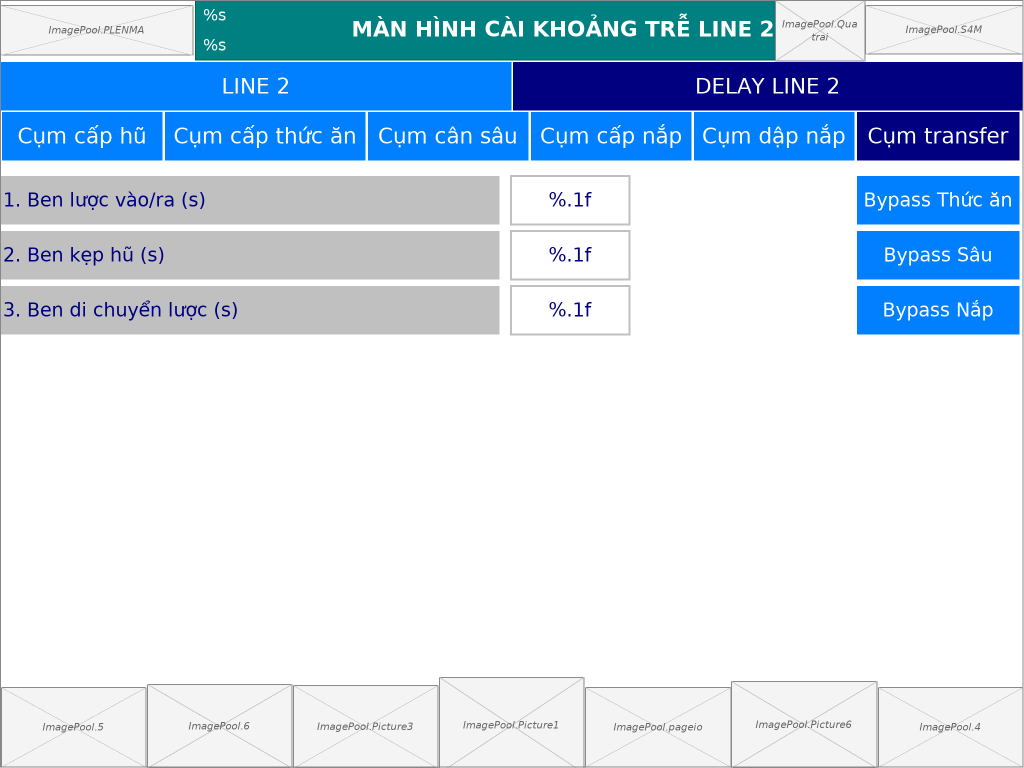
VISUALIZATION N_Setting_Delay_Tranfer2  // 1024x768
    Frame (0,687 1024x80)
        shows N_Footer_Line2()
    Frame (0,0 1024x60)
        shows N_Header()
    Textfield (353,4 420x50), "MÀN HÌNH CÀI KHOẢNG TRỄ LINE 2"
    Rectangle (0,175 500x50), "1. Ben lược vào/ra (s)"
    Rectangle (0,230 500x50), "2. Ben kẹp hũ (s)"
    Rectangle (0,285 500x50), "3. Ben di chuyển lược (s)"
    Group (0,61 1023x100)
        Rectangle (0,0 512x50), "LINE 2"
            OnMouseClick: change screen: N_Setting_Line2
        Rectangle (1,50 162x50), "Cụm cấp hũ"
            OnMouseClick: change screen: N_Setting_Delay_JarSupply2
        Rectangle (164,50 202x50), "Cụm cấp thức ăn"
            OnMouseClick: change screen: N_Setting_Delay_FoodSupply2
        Rectangle (367,50 162x50), "Cụm cân sâu"
            OnMouseClick: change screen: N_Setting_Delay_WorwWeight2
        Rectangle (530,50 162x50), "Cụm cấp nắp"
            OnMouseClick: change screen: N_Setting_Delay_LidSupply2
        Rectangle (693,50 162x50), "Cụm dập nắp"
            OnMouseClick: change screen: N_Setting_Delay_LidPressing2
        Rectangle (856,50 164x50), "Cụm transfer"
            OnMouseClick: change screen: N_Setting_Delay_Tranfer2
        Rectangle (512,0 511x50), "DELAY LINE 2"
            OnMouseClick: change screen: N_Setting_Delay_JarSupply2
    Image (775,0 90x61), image: ImagePool.Qua trai
        OnMouseClick: change screen: N_Setting_Delay_Tranfer1
    Rectangle (510,175 120x50), "%.1f", text variable: PR_Line02.fTimer_Comb
        OnMouseClick: write PR_Line02.fTimer_Comb via VisuDialogs.Numpad
    Rectangle (510,230 120x50), "%.1f", text variable: PR_Line02.fTimer_Clip
        OnMouseClick: write PR_Line02.fTimer_Clip via VisuDialogs.Numpad
    Rectangle (510,285 120x50), "%.1f", text variable: PR_Line02.fTimer_Move_Comb
        OnMouseClick: write PR_Line02.fTimer_Move_Comb via VisuDialogs.Numpad
    Rectangle (856,175 164x50), "Bypass Thức ăn"
        toggle PR_Line02.bypassFood
    Rectangle (856,230 164x50), "Bypass Sâu"
        toggle PR_Line02.bypassWorm
    Rectangle (856,285 164x50), "Bypass Nắp"
        toggle PR_Line02.bypassLid
END_VISUALIZATION

// ---- VISUs/Setting/N_Setting_Delay_WormWeight1.TcVIS
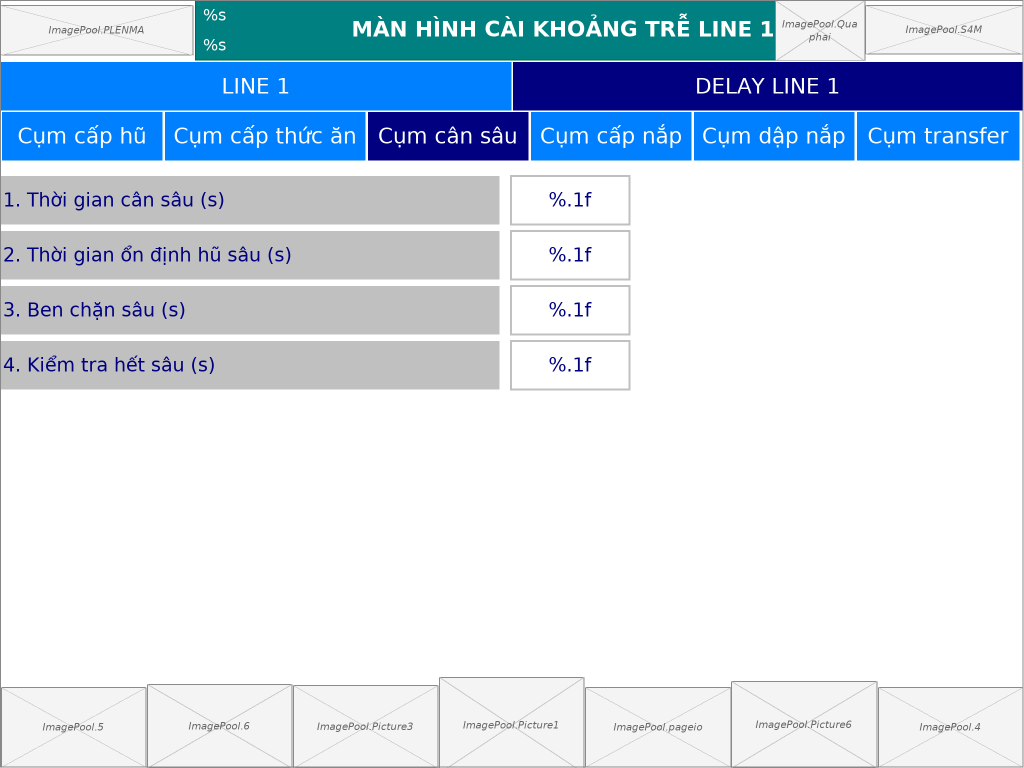
VISUALIZATION N_Setting_Delay_WormWeight1  // 1024x768
    Frame (0,687 1024x80)
        shows N_Footer_Line1()
    Frame (0,0 1024x60)
        shows N_Header()
    Textfield (353,4 420x50), "MÀN HÌNH CÀI KHOẢNG TRỄ LINE 1"
    Rectangle (0,61 512x50), "LINE 1"
        OnMouseClick: change screen: N_Setting_Line1
    Image (775,0 90x61), image: ImagePool.Qua phai
        OnMouseClick: change screen: N_Setting_Delay_WorwWeight2
    Rectangle (0,175 500x50), "1. Thời gian cân sâu (s)"
    Rectangle (0,285 500x50), "3. Ben chặn sâu (s)"
    Rectangle (510,285 120x50), "%.1f", text variable: PR_Line01.fTimer_Check_Cylinder
        OnMouseClick: write PR_Line01.fTimer_Check_Cylinder via VisuDialogs.Numpad
    Rectangle (510,230 120x50), "%.1f", text variable: PR_Line01.fTimer_Worm
        OnMouseClick: write PR_Line01.fTimer_Worm via VisuDialogs.Numpad
    Rectangle (0,230 500x50), "2. Thời gian ổn định hũ sâu (s)"
    Rectangle (510,175 120x50), "%.1f", text variable: PR_Line01.fTimer_Alarm_Worm
        OnMouseClick: write PR_Line01.fTimer_Alarm_Worm via VisuDialogs.Numpad
    Rectangle (1,111 162x50), "Cụm cấp hũ"
        OnMouseClick: change screen: N_Setting_Delay_JarSupply1
    Rectangle (164,111 202x50), "Cụm cấp thức ăn"
        OnMouseClick: change screen: N_Setting_Delay_FoodSupply1
    Rectangle (367,111 162x50), "Cụm cân sâu"
        OnMouseClick: change screen: N_Setting_Delay_WormWeight1
    Rectangle (530,111 162x50), "Cụm cấp nắp"
        OnMouseClick: change screen: N_Setting_Delay_LidSupply1
    Rectangle (693,111 162x50), "Cụm dập nắp"
        OnMouseClick: change screen: N_Setting_Delay_LidPressing1
    Rectangle (856,111 164x50), "Cụm transfer"
        OnMouseClick: change screen: N_Setting_Delay_Tranfer1
    Rectangle (512,61 511x50), "DELAY LINE 1"
        OnMouseClick: change screen: N_Setting_Delay_JarSupply1
    Rectangle (0,340 500x50), "4. Kiểm tra hết sâu (s)"
    Rectangle (510,340 120x50), "%.1f", text variable: PR_Line01.fTimer_Error_Worm
        OnMouseClick: write PR_Line01.fTimer_Error_Worm via VisuDialogs.Numpad
END_VISUALIZATION

// ---- VISUs/Setting/N_Setting_Delay_WorwWeight2.TcVIS
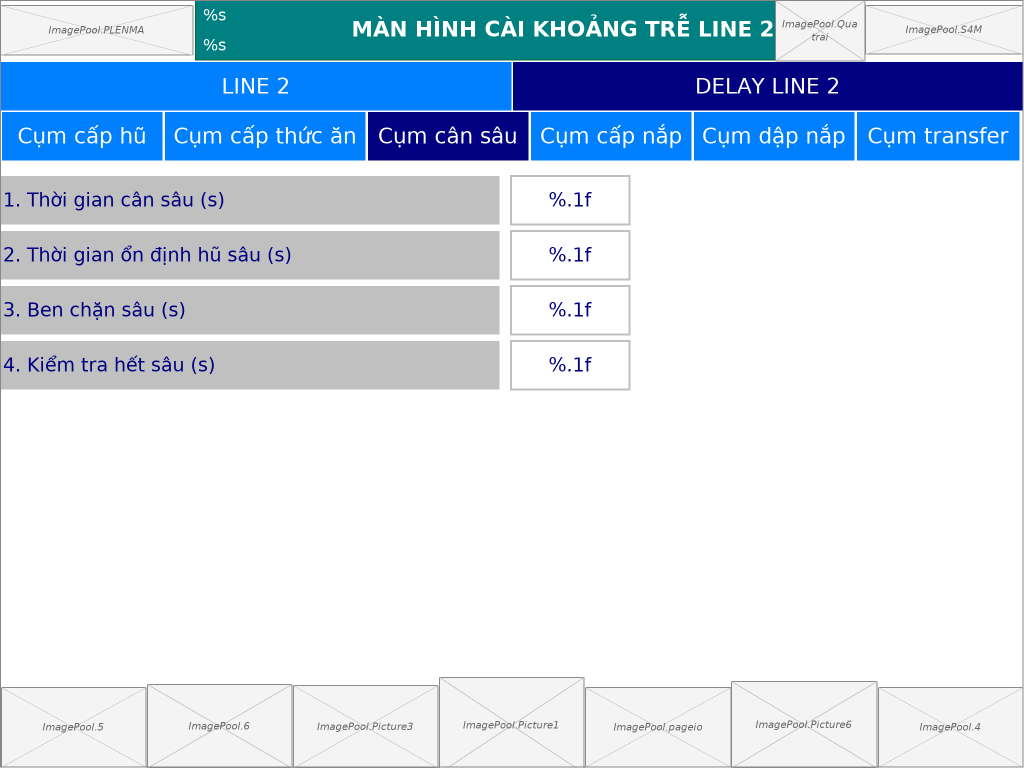
VISUALIZATION N_Setting_Delay_WorwWeight2  // 1024x768
    Frame (0,687 1024x80)
        shows N_Footer_Line2()
    Frame (0,0 1024x60)
        shows N_Header()
    Textfield (353,4 420x50), "MÀN HÌNH CÀI KHOẢNG TRỄ LINE 2"
    Rectangle (0,175 500x50), "1. Thời gian cân sâu (s)"
    Rectangle (0,285 500x50), "3. Ben chặn sâu (s)"
    Rectangle (0,230 500x50), "2. Thời gian ổn định hũ sâu (s)"
    Rectangle (0,61 512x50), "LINE 2"
        OnMouseClick: change screen: N_Setting_Line2
    Rectangle (1,111 162x50), "Cụm cấp hũ"
        OnMouseClick: change screen: N_Setting_Delay_JarSupply2
    Rectangle (164,111 202x50), "Cụm cấp thức ăn"
        OnMouseClick: change screen: N_Setting_Delay_FoodSupply2
    Rectangle (367,111 162x50), "Cụm cân sâu"
        OnMouseClick: change screen: N_Setting_Delay_WorwWeight2
    Rectangle (530,111 162x50), "Cụm cấp nắp"
        OnMouseClick: change screen: N_Setting_Delay_LidSupply2
    Rectangle (693,111 162x50), "Cụm dập nắp"
        OnMouseClick: change screen: N_Setting_Delay_LidPressing2
    Rectangle (856,111 164x50), "Cụm transfer"
        OnMouseClick: change screen: N_Setting_Delay_Tranfer2
    Rectangle (512,61 511x50), "DELAY LINE 2"
        OnMouseClick: change screen: N_Setting_Delay_JarSupply2
    Image (775,0 90x61), image: ImagePool.Qua trai
        OnMouseClick: change screen: N_Setting_Delay_WormWeight1
    Rectangle (510,285 120x50), "%.1f", text variable: PR_Line02.fTimer_Check_Cylinder
        OnMouseClick: write PR_Line02.fTimer_Check_Cylinder via VisuDialogs.Numpad
    Rectangle (510,230 120x50), "%.1f", text variable: PR_Line02.fTimer_Worm
        OnMouseClick: write PR_Line02.fTimer_Worm via VisuDialogs.Numpad
    Rectangle (510,175 120x50), "%.1f", text variable: PR_Line02.fTimer_Alarm_Worm
        OnMouseClick: write PR_Line02.fTimer_Alarm_Worm via VisuDialogs.Numpad
    Rectangle (0,340 500x50), "4. Kiểm tra hết sâu (s)"
    Rectangle (510,340 120x50), "%.1f", text variable: PR_Line02.fTimer_Error_Worm
        OnMouseClick: write PR_Line02.fTimer_Error_Worm via VisuDialogs.Numpad
END_VISUALIZATION

// ---- VISUs/Setting/N_Setting_Line1.TcVIS
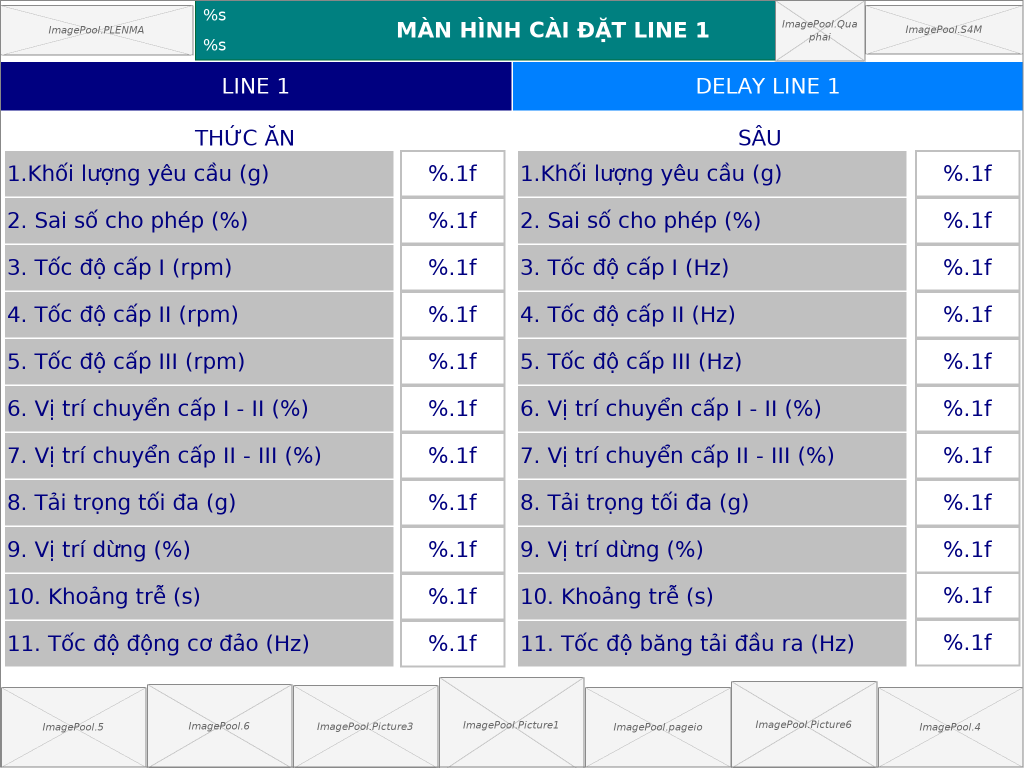
VISUALIZATION N_Setting_Line1  // 1024x768
    Rectangle (512,61 512x50), "DELAY LINE 1"
        OnMouseClick: change screen: N_Setting_Delay_JarSupply1
    Frame (0,687 1024x80)
        shows N_Footer_Line1()
    Frame (0,0 1024x60)
        shows N_Header()
    Textfield (353,5 400x50), "MÀN HÌNH CÀI ĐẶT LINE 1"
    Textfield (170,120 150x36), "THỨC ĂN"
    Textfield (720,120 80x36), "SÂU"
    Rectangle (0,61 512x50), "LINE 1"
        OnMouseClick: change screen: N_Setting_Line1
    Rectangle (517,150 390x47), "1.Khối lượng yêu cầu (g)"
    Rectangle (517,197 390x47), "2. Sai số cho phép (%)"
    Rectangle (517,244 390x47), "3. Tốc độ cấp I (Hz)"
    Rectangle (517,291 390x47), "4. Tốc độ cấp II (Hz)"
    Rectangle (517,385 390x47), "6. Vị trí chuyển cấp I - II (%)"
    Rectangle (517,479 390x47), "8. Tải trọng tối đa (g)"
    Rectangle (517,338 390x47), "5. Tốc độ cấp III (Hz)"
    Rectangle (517,432 390x47), "7. Vị trí chuyển cấp II - III (%)"
    Rectangle (517,573 390x47), "10. Khoảng trễ (s)"
    Rectangle (517,526 390x47), "9. Vị trí dừng (%)"
    Textfield (915,150 105x47), "%.1f", text variable: PR_Line01.fDerisedWeight_Worm
        OnMouseClick: write PR_Line01.fDerisedWeight_Worm via VisuDialogs.Numpad
    Textfield (915,197 105x47), "%.1f", text variable: PR_Line01.fDelta_Worm
        OnMouseClick: write PR_Line01.fDelta_Worm via VisuDialogs.Numpad
    Textfield (915,244 105x47), "%.1f", text variable: PR_Line01.fFast_Speed_vibrating_funnel
        OnMouseClick: write PR_Line01.fFast_Speed_vibrating_funnel via VisuDialogs.Numpad
    Textfield (915,291 105x47), "%.1f", text variable: PR_Line01.fSlow_Speed_vibrating_funnel_1
        OnMouseClick: write PR_Line01.fSlow_Speed_vibrating_funnel_1 via VisuDialogs.Numpad
    Textfield (915,338 105x47), "%.1f", text variable: PR_Line01.fSlow_Speed_vibrating_funnel_2
        OnMouseClick: write PR_Line01.fSlow_Speed_vibrating_funnel_2 via VisuDialogs.Numpad
    Textfield (915,385 105x47), "%.1f", text variable: PR_Line01.fChangeMode_Worm_1
        OnMouseClick: write PR_Line01.fChangeMode_Worm_1 via VisuDialogs.Numpad
    Textfield (915,432 105x47), "%.1f", text variable: PR_Line01.fChangeMode_Worm_2
        OnMouseClick: write PR_Line01.fChangeMode_Worm_2 via VisuDialogs.Numpad
    Textfield (915,479 105x47), "%.1f", text variable: PR_Line01.fMaxWeight_Worm
        OnMouseClick: write PR_Line01.fMaxWeight_Worm via VisuDialogs.Numpad
    Textfield (915,526 105x47), "%.1f", text variable: PR_Line01.fPerStop_Worm
        OnMouseClick: write PR_Line01.fPerStop_Worm via VisuDialogs.Numpad
    Textfield (915,572 105x47), "%.1f", text variable: PR_Line01.fTimer_Check_Worm
        OnMouseClick: write PR_Line01.fTimer_Check_Worm via VisuDialogs.Numpad
    Rectangle (4,150 390x47), "1.Khối lượng yêu cầu (g)"
    Rectangle (4,197 390x47), "2. Sai số cho phép (%)"
    Rectangle (4,244 390x47), "3. Tốc độ cấp I (rpm)"
    Rectangle (4,291 390x47), "4. Tốc độ cấp II (rpm)"
    Rectangle (4,385 390x47), "6. Vị trí chuyển cấp I - II (%)"
    Rectangle (4,479 390x47), "8. Tải trọng tối đa (g)"
    Rectangle (4,338 390x47), "5. Tốc độ cấp III (rpm)"
    Rectangle (4,432 390x47), "7. Vị trí chuyển cấp II - III (%)"
    Rectangle (4,573 390x47), "10. Khoảng trễ (s)"
    Rectangle (4,526 390x47), "9. Vị trí dừng (%)"
    Rectangle (4,620 390x47), "11. Tốc độ động cơ đảo (Hz)"
    Textfield (400,150 105x47), "%.1f", text variable: PR_Line01.fDerisedWeight_Food
        OnMouseClick: write PR_Line01.fDerisedWeight_Food via VisuDialogs.Numpad
    Textfield (400,197 105x47), "%.1f", text variable: PR_Line01.fDelta_Food
        OnMouseClick: write PR_Line01.fDelta_Food via VisuDialogs.Numpad
    Textfield (400,244 105x47), "%.1f", text variable: PR_Line01.fFast_Speed
        OnMouseClick: write PR_Line01.fFast_Speed via VisuDialogs.Numpad
    Textfield (400,291 105x47), "%.1f", text variable: PR_Line01.fSlow_Speed_1
        OnMouseClick: write PR_Line01.fSlow_Speed_1 via VisuDialogs.Numpad
    Textfield (400,338 105x47), "%.1f", text variable: PR_Line01.fSlow_Speed_2
        OnMouseClick: write PR_Line01.fSlow_Speed_2 via VisuDialogs.Numpad
    Textfield (400,385 105x47), "%.1f", text variable: PR_Line01.fChangeMode_Food_1
        OnMouseClick: write PR_Line01.fChangeMode_Food_1 via VisuDialogs.Numpad
    Textfield (400,432 105x47), "%.1f", text variable: PR_Line01.fChangeMode_Food_2
        OnMouseClick: write PR_Line01.fChangeMode_Food_2 via VisuDialogs.Numpad
    Textfield (400,479 105x47), "%.1f", text variable: PR_Line01.fMaxWeight_Food
        OnMouseClick: write PR_Line01.fMaxWeight_Food via VisuDialogs.Numpad
    Textfield (400,526 105x47), "%.1f", text variable: PR_Line01.fPerStop_Food
        OnMouseClick: write PR_Line01.fPerStop_Food via VisuDialogs.Numpad
    Textfield (400,573 105x47), "%.1f", text variable: PR_Line01.fTimer_Check_Food
        OnMouseClick: write PR_Line01.fTimer_Check_Food via VisuDialogs.Numpad
    Textfield (400,620 105x47), "%.1f", text variable: PR_Line01.fSpeed_motor_mixer
        OnMouseClick: write PR_Line01.fSpeed_motor_mixer via VisuDialogs.Numpad
    Image (775,0 90x61), image: ImagePool.Qua phai
        OnMouseClick: change screen: N_Setting_Line2
    Rectangle (517,620 390x47), "11. Tốc độ băng tải đầu ra (Hz)"
    Textfield (915,619 105x47), "%.1f", text variable: PR_Conveyor_Out.fSpeed_Conveyor
        OnMouseClick: write PR_Conveyor_Out.fSpeed_Conveyor via VisuDialogs.Numpad
END_VISUALIZATION

// ---- VISUs/Setting/N_Setting_Line2.TcVIS
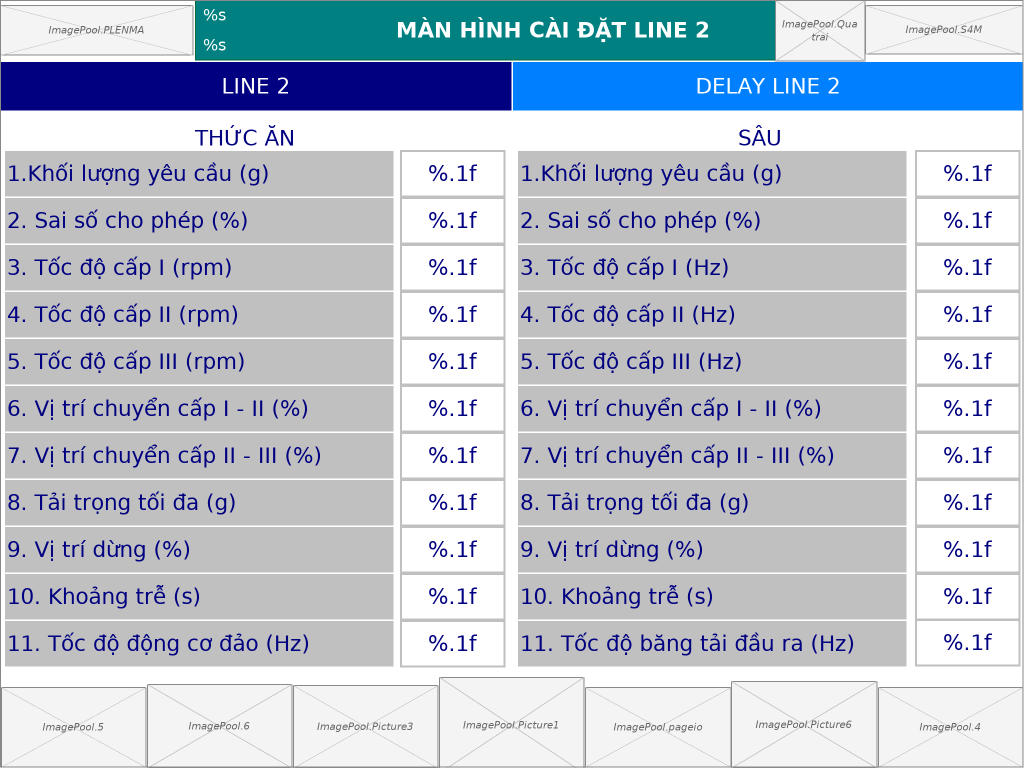
VISUALIZATION N_Setting_Line2  // 1024x768
    Frame (0,687 1024x80)
        shows N_Footer_Line2()
    Frame (0,0 1024x60)
        shows N_Header()
    Textfield (353,5 400x50), "MÀN HÌNH CÀI ĐẶT LINE 2"
    Textfield (170,120 150x36), "THỨC ĂN"
    Textfield (720,120 80x36), "SÂU"
    Rectangle (0,61 512x50), "LINE 2"
        OnMouseClick: change screen: N_Setting_Line2
    Rectangle (512,61 512x50), "DELAY LINE 2"
        OnMouseClick: change screen: N_Setting_Delay_JarSupply2
    Rectangle (517,150 390x47), "1.Khối lượng yêu cầu (g)"
    Rectangle (517,197 390x47), "2. Sai số cho phép (%)"
    Rectangle (517,244 390x47), "3. Tốc độ cấp I (Hz)"
    Rectangle (517,291 390x47), "4. Tốc độ cấp II (Hz)"
    Rectangle (517,385 390x47), "6. Vị trí chuyển cấp I - II (%)"
    Rectangle (517,479 390x47), "8. Tải trọng tối đa (g)"
    Rectangle (517,338 390x47), "5. Tốc độ cấp III (Hz)"
    Rectangle (517,432 390x47), "7. Vị trí chuyển cấp II - III (%)"
    Rectangle (517,573 390x47), "10. Khoảng trễ (s)"
    Rectangle (517,526 390x47), "9. Vị trí dừng (%)"
    Textfield (915,150 105x47), "%.1f", text variable: PR_Line02.fDerisedWeight_Worm
        OnMouseClick: write PR_Line02.fDerisedWeight_Worm via VisuDialogs.Numpad
    Textfield (915,197 105x47), "%.1f", text variable: PR_Line02.fDelta_Worm
        OnMouseClick: write PR_Line02.fDelta_Worm via VisuDialogs.Numpad
    Textfield (915,244 105x47), "%.1f", text variable: PR_Line02.fFast_Speed_vibrating_funnel
        OnMouseClick: write PR_Line02.fFast_Speed_vibrating_funnel via VisuDialogs.Numpad
    Textfield (915,291 105x47), "%.1f", text variable: PR_Line02.fSlow_Speed_vibrating_funnel_1
        OnMouseClick: write PR_Line02.fSlow_Speed_vibrating_funnel_1 via VisuDialogs.Numpad
    Textfield (915,338 105x47), "%.1f", text variable: PR_Line02.fSlow_Speed_vibrating_funnel_2
        OnMouseClick: write PR_Line02.fSlow_Speed_vibrating_funnel_2 via VisuDialogs.Numpad
    Textfield (915,385 105x47), "%.1f", text variable: PR_Line02.fChangeMode_Worm_1
        OnMouseClick: write PR_Line02.fChangeMode_Worm_1 via VisuDialogs.Numpad
    Textfield (915,432 105x47), "%.1f", text variable: PR_Line02.fChangeMode_Worm_2
        OnMouseClick: write PR_Line02.fChangeMode_Worm_2 via VisuDialogs.Numpad
    Textfield (915,479 105x47), "%.1f", text variable: PR_Line02.fMaxWeight_Worm
        OnMouseClick: write PR_Line02.fMaxWeight_Worm via VisuDialogs.Numpad
    Textfield (915,526 105x47), "%.1f", text variable: PR_Line02.fPerStop_Worm
        OnMouseClick: write PR_Line02.fPerStop_Worm via VisuDialogs.Numpad
    Textfield (915,573 105x47), "%.1f", text variable: PR_Line02.fTimer_Check_Worm
        OnMouseClick: write PR_Line02.fTimer_Check_Worm via VisuDialogs.Numpad
    Rectangle (4,150 390x47), "1.Khối lượng yêu cầu (g)"
    Rectangle (4,197 390x47), "2. Sai số cho phép (%)"
    Rectangle (4,244 390x47), "3. Tốc độ cấp I (rpm)"
    Rectangle (4,291 390x47), "4. Tốc độ cấp II (rpm)"
    Rectangle (4,385 390x47), "6. Vị trí chuyển cấp I - II (%)"
    Rectangle (4,479 390x47), "8. Tải trọng tối đa (g)"
    Rectangle (4,338 390x47), "5. Tốc độ cấp III (rpm)"
    Rectangle (4,432 390x47), "7. Vị trí chuyển cấp II - III (%)"
    Rectangle (4,573 390x47), "10. Khoảng trễ (s)"
    Rectangle (4,526 390x47), "9. Vị trí dừng (%)"
    Rectangle (4,620 390x47), "11. Tốc độ động cơ đảo (Hz)"
    Textfield (400,150 105x47), "%.1f", text variable: PR_Line02.fDerisedWeight_Food
        OnMouseClick: write PR_Line02.fDerisedWeight_Food via VisuDialogs.Numpad
    Textfield (400,197 105x47), "%.1f", text variable: PR_Line02.fDelta_Food
        OnMouseClick: write PR_Line02.fDelta_Food via VisuDialogs.Numpad
    Textfield (400,244 105x47), "%.1f", text variable: PR_Line02.fFast_Speed
        OnMouseClick: write PR_Line02.fFast_Speed via VisuDialogs.Numpad
    Textfield (400,291 105x47), "%.1f", text variable: PR_Line02.fSlow_Speed_1
        OnMouseClick: write PR_Line02.fSlow_Speed_1 via VisuDialogs.Numpad
    Textfield (400,338 105x47), "%.1f", text variable: PR_Line02.fSlow_Speed_2
        OnMouseClick: write PR_Line02.fSlow_Speed_2 via VisuDialogs.Numpad
    Textfield (400,385 105x47), "%.1f", text variable: PR_Line02.fChangeMode_Food_1
        OnMouseClick: write PR_Line02.fChangeMode_Food_1 via VisuDialogs.Numpad
    Textfield (400,432 105x47), "%.1f", text variable: PR_Line02.fChangeMode_Food_2
        OnMouseClick: write PR_Line02.fChangeMode_Food_2 via VisuDialogs.Numpad
    Textfield (400,479 105x47), "%.1f", text variable: PR_Line02.fMaxWeight_Food
        OnMouseClick: write PR_Line02.fMaxWeight_Food via VisuDialogs.Numpad
    Textfield (400,526 105x47), "%.1f", text variable: PR_Line02.fPerStop_Food
        OnMouseClick: write PR_Line02.fPerStop_Food via VisuDialogs.Numpad
    Textfield (400,573 105x47), "%.1f", text variable: PR_Line02.fTimer_Check_Food
        OnMouseClick: write PR_Line02.fTimer_Check_Food via VisuDialogs.Numpad
    Textfield (400,620 105x47), "%.1f", text variable: PR_Line02.fSpeed_motor_mixer
        OnMouseClick: write PR_Line02.fSpeed_motor_mixer via VisuDialogs.Numpad
    Image (775,0 90x61), image: ImagePool.Qua trai
        OnMouseClick: change screen: N_Setting_Line1
    Rectangle (517,620 390x47), "11. Tốc độ băng tải đầu ra (Hz)"
    Textfield (915,619 105x47), "%.1f", text variable: PR_Conveyor_Out.fSpeed_Conveyor
        OnMouseClick: write PR_Conveyor_Out.fSpeed_Conveyor via VisuDialogs.Numpad
END_VISUALIZATION

// ---- VISUs/Title/N_Footer_Alarm.TcVIS
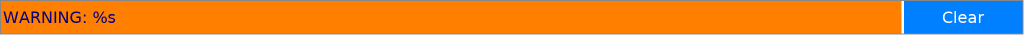
VISUALIZATION N_Footer_Alarm  // 1024x35
    Rectangle (0,0 902x35), "WARNING: %s", text variable: stWarningTxt1, invisible if: not bWrn2, input disabled if: not bWrn2
    Rectangle (0,0 902x35), "WARNING: %s", text variable: stWarningTxt, invisible if: not bWrn, input disabled if: not bWrn
    Rectangle (903,0 120x35), "Clear", invisible if: not bxoa, input disabled if: not bxoa
        OnMouseDown: execute {
            bWrn := FALSE;
            bWrn2 := FALSE;
            bWarning := FALSE;
            bWarning2 := FALSE;
            bxoa := FALSE;
            bSirens := false;
        }
END_VISUALIZATION

// ---- VISUs/Title/N_Footer_Alarm_1.TcVIS
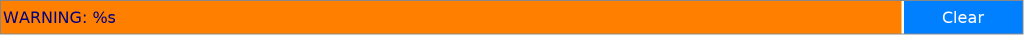
VISUALIZATION N_Footer_Alarm_1  // 1024x35
    Rectangle (0,-1 902x35), "WARNING: %s", text variable: stWarningTxt2, invisible if: not bWrn, input disabled if: not bWrn
    Rectangle (0,0 902x35), "WARNING: %s", text variable: StWarningTxt3, invisible if: not bWrn2, input disabled if: not bWrn2
    Rectangle (903,0 120x35), "Clear", invisible if: not bxoa, input disabled if: not bxoa
        OnMouseDown: execute {
            bWrn := FALSE;
            bWrn2 := FALSE;
            bWarning := FALSE;
            bWarning2 := FALSE;
            bxoa := FALSE;
        }
END_VISUALIZATION

// ---- VISUs/Title/N_Footer_Line1.TcVIS
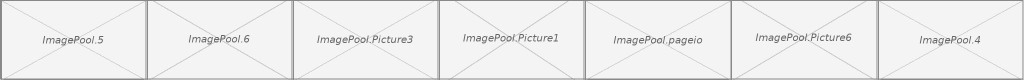
VISUALIZATION N_Footer_Line1  // 1024x80
    Image (878,0 145x80), invisible if: GVL_OF_VU.bVN, input disabled if: GVL_OF_VU.bVN, image: ImagePool.3
        OnMouseDown: ChangeLanguage ChangeLanguage=vn
    Image (878,0 145x80), invisible if: not GVL_OF_VU.bVN, input disabled if: not GVL_OF_VU.bVN, image: ImagePool.4
        OnMouseDown: ChangeLanguage ChangeLanguage=eng
    Image (1,0 145x80), input disabled if: not bResetmanual1, image: ImagePool.5
        OnMouseDown: change screen: MAIN_LINE1
        OnMouseDown: execute {
            MAIN.bModeAuto := TRUE;
            MAIN.bModeManual := FALSE;
            bWriteData := TRUE;
        }
    Image (147,-3 145x84), input disabled if: bResetAuto1, image: ImagePool.6
        OnMouseClick: change screen: N_JarSupply1
        OnMouseClick: execute {
            MAIN.bModeManual := TRUE;
            MAIN.bModeAuto := FALSE;
            bWriteData := TRUE;
        }
    Image (293,-2 145x83), image: ImagePool.Picture3
        OnMouseClick: change screen: N_Setting_Line1
    Image (439,-10 145x96), image: ImagePool.Picture1
        OnMouseClick: change screen: N_Recipe_Line1
    Image (585,0 146x80), image: ImagePool.pageio
        OnMouseClick: change screen: N_PLC_I1
    Image (731,-6 146x87), image: ImagePool.Picture6
        OnMouseClick: change screen: N_Alarm
END_VISUALIZATION

// ---- VISUs/Title/N_Footer_Line2.TcVIS
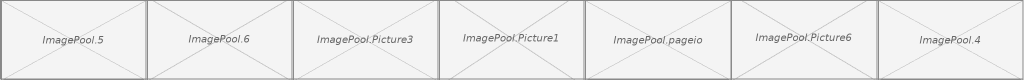
VISUALIZATION N_Footer_Line2  // 1024x80
    Image (1,0 145x80), input disabled if: Not bResetmanual2, image: ImagePool.5
        OnMouseDown: change screen: MAIN_LINE2
        OnMouseDown: execute { MAIN_LINE2.bModeAuto := TRUE; MAIN_LINE2.bModeManual := FALSE; }
    Image (147,-3 145x84), input disabled if: bResetAuto2, image: ImagePool.6
        OnMouseDown: change screen: N_JarSupply2
        OnMouseDown: execute { MAIN_LINE2.bModeManual := TRUE; MAIN_LINE2.bModeAuto := FALSE; }
    Image (293,-2 145x83), image: ImagePool.Picture3
        OnMouseClick: change screen: N_Setting_Line2
    Image (439,-10 145x96), image: ImagePool.Picture1
        OnMouseClick: change screen: N_Recipe_Line2
    Image (585,0 146x80), image: ImagePool.pageio
        OnMouseClick: change screen: N_PLC_I2
    Image (731,-6 146x87), image: ImagePool.Picture6
        OnMouseClick: change screen: N_Alarm_1
    Image (878,0 145x80), invisible if: GVL_OF_VU.bVN, input disabled if: GVL_OF_VU.bVN, image: ImagePool.3
        OnMouseDown: ChangeLanguage ChangeLanguage=vn
    Image (878,0 145x80), invisible if: not GVL_OF_VU.bVN, input disabled if: not GVL_OF_VU.bVN, image: ImagePool.4
        OnMouseDown: ChangeLanguage ChangeLanguage=eng
END_VISUALIZATION

// ---- VISUs/Title/N_Header.TcVIS
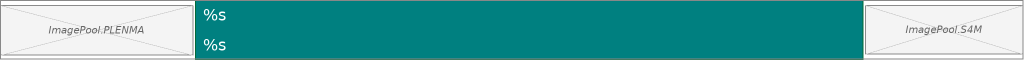
VISUALIZATION N_Header  // 1024x60
    Image (0,5 193x50), image: ImagePool.PLENMA
        OnMouseClick: VisuUserMgmt Type=Logout
    Image (865,5 158x49), image: ImagePool.S4M
    Rectangle (195,0 668x60)
    Textfield (200,0 150x30), "%s", text variable: Onlyday
    Textfield (200,30 150x30), "%s", text variable: OnlyTime
END_VISUALIZATION

// ---- VISUs/Title/N_Login.TcVIS
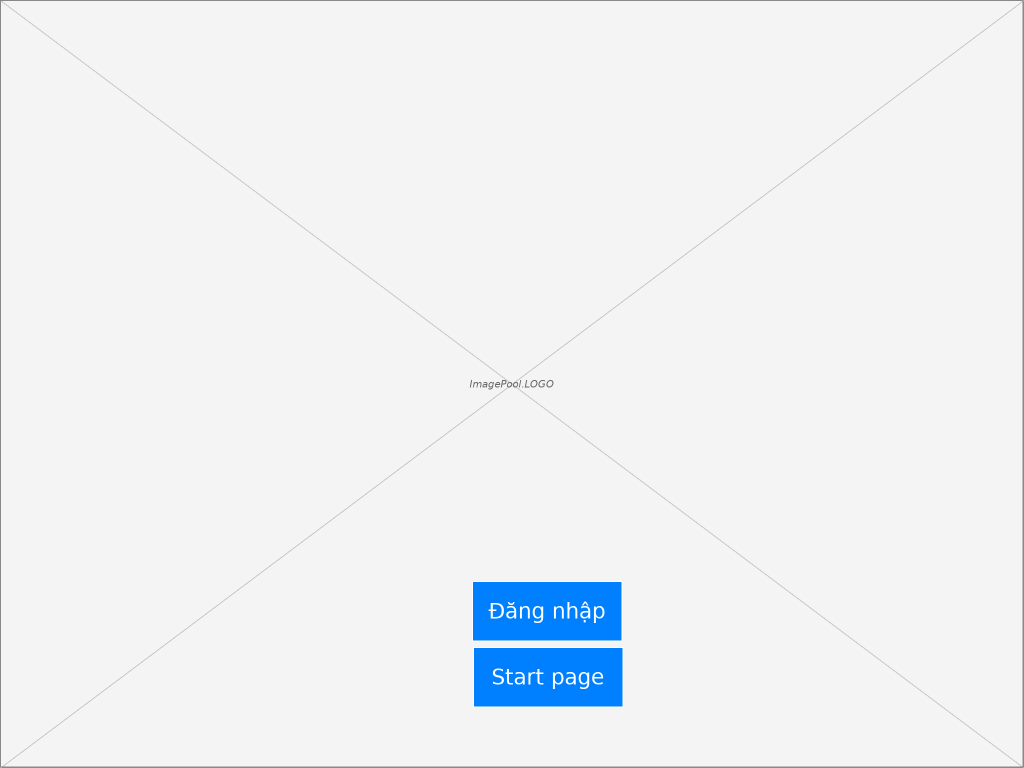
VISUALIZATION N_Login  // 1024x768
    Image (0,0 1024x768), image: ImagePool.LOGO
    Rectangle (472,581 150x60), "Đăng nhập"
        OnMouseDown: VisuUserMgmt Type=Login
    Rectangle (473,647 150x60), "Start page"
        OnMouseDown: execute { username := ''; }
        OnMouseDown: OpenDialog Dialog=startpage, OpenModal=True, OpenCentered=True
END_VISUALIZATION

// ---- VISUs/Title/startpage.TcVIS
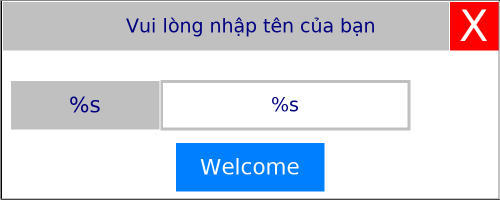
VISUALIZATION startpage  // 500x200
    Rectangle (1,0 500x200)
    Rectangle (2,1 498x50), "Vui lòng nhập tên của bạn"
    Rectangle (160,80 250x50), "%s", text variable: username
        OnMouseDown: write username via VisuDialogs.Keypad
    Rectangle (175,142 150x50), "Welcome", invisible if: not openstartpage, input disabled if: not openstartpage
        OnMouseDown: CloseDialog Dialog=startpage, Result=OK, NumpadKeypadSet=True
        OnMouseDown: change screen: N_Setting_Line1
    Rectangle (449,1 50x50), "X"
        OnMouseDown: CloseDialog Dialog=startpage, Result=OK, NumpadKeypadSet=True
    Rectangle (10,80 150x50), "%s", text variable: getuser
END_VISUALIZATION
